LIN {X 0,Y 361.852,Z 288.032,A -85,B 0,C 180,E1 -12933.467,E2 -12933.467} C_VEL
LIN {X 0,Y 361.859,Z 288.029,A -85,B 0,C 180,E1 -12937.142,E2 -12937.142} C_VEL
LIN {X 0,Y 361.84,Z 288.029,A -85,B 0,C 180,E1 -12940.72,E2 -12940.72} C_VEL
LIN {X 0,Y 361.875,Z 288.032,A -85,B 0,C 180,E1 -12943.063,E2 -12943.063} C_VEL
LIN {X 0,Y 361.997,Z 288.011,A -85,B 0,C 180,E1 -12946.528,E2 -12946.528} C_VEL
LIN {X 0,Y 361.996,Z 288.014,A -85,B 0,C 180,E1 -12949.937,E2 -12949.937} C_VEL
LIN {X 0,Y 362.116,Z 288.001,A -85,B 0,C 180,E1 -12953.313,E2 -12953.313} C_VEL
LIN {X 0,Y 362.269,Z 287.981,A -85,B 0,C 180,E1 -12957.776,E2 -12957.776} C_VEL
LIN {X 0,Y 362.265,Z 287.979,A -85,B 0,C 180,E1 -12962.224,E2 -12962.224} C_VEL
LIN {X 0,Y 362.122,Z 287.997,A -85,B 0,C 180,E1 -12966.687,E2 -12966.687} C_VEL
LIN {X 0,Y 361.998,Z 288.011,A -85,B 0,C 180,E1 -12970.063,E2 -12970.063} C_VEL
LIN {X 0,Y 361.996,Z 288.018,A -85,B 0,C 180,E1 -12973.899,E2 -12973.899} C_VEL
LIN {X 0,Y 361.966,Z 288.024,A -85,B 0,C 180,E1 -12977.939,E2 -12977.939} C_VEL
LIN {X 0,Y 361.89,Z 288.034,A -85,B 0,C 180,E1 -12981.653,E2 -12981.653} C_VEL
LIN {X 0,Y 361.889,Z 288.003,A -85,B 0,C 180,E1 -12985.293,E2 -12985.293} C_VEL
LIN {X 0,Y 361.853,Z 288.035,A -85,B 0,C 180,E1 -12989.074,E2 -12989.074} C_VEL
LIN {X 0,Y 361.848,Z 288.021,A -85,B 0,C 180,E1 -12992.945,E2 -12992.945} C_VEL
LIN {X 0,Y 361.866,Z 288.032,A -85,B 0,C 180,E1 -12995.637,E2 -12995.637} C_VEL
LIN {X 0,Y 361.868,Z 288.029,A -85,B 0,C 180,E1 -12999.027,E2 -12999.027} C_VEL
LIN {X 0,Y 361.834,Z 288.037,A -85,B 0,C 180,E1 -13002.829,E2 -13002.829} C_VEL
LIN {X 0,Y 361.816,Z 288.04,A -85,B 0,C 180,E1 -13005.947,E2 -13005.947} C_VEL
LIN {X 0,Y 361.833,Z 288.027,A -85,B 0,C 180,E1 -13009.245,E2 -13009.245} C_VEL
LIN {X 0,Y 361.889,Z 288.094,A -85,B 0,C 180,E1 -13012.392,E2 -13012.392} C_VEL
LIN {X 0,Y 365.714,Z 301.841,A -85,B 0,C 180,E1 -13015.724,E2 -13015.724} C_VEL
LIN {X 0,Y 368.692,Z 314.163,A -85,B 0,C 180,E1 -13018.496,E2 -13018.496} C_VEL
LIN {X 0,Y 373.915,Z 326.027,A -85,B 0,C 180,E1 -13019.24,E2 -13019.24} C_VEL
LIN {X 0,Y 378.235,Z 348.319,A -85,B 0,C 180,E1 -13020.103,E2 -13020.103} C_VEL
LIN {X 0,Y 380.008,Z 359.01,A -85,B 0,C 180,E1 -13020.482,E2 -13020.482} C_VEL
LIN {X 0,Y 377.135,Z 474.361,A -85,B 0,C 180,E1 -13022.685,E2 -13022.685} C_VEL
LIN {X 0,Y 376.476,Z 489.459,A -85,B 0,C 180,E1 -13023.084,E2 -13023.084} C_VEL
LIN {X 0,Y 375.293,Z 504.296,A -85,B 0,C 180,E1 -13023.667,E2 -13023.667} C_VEL
LIN {X 0,Y 373.914,Z 518.628,A -85,B 0,C 180,E1 -13024.448,E2 -13024.448} C_VEL
LIN {X 0,Y 372.271,Z 532.938,A -85,B 0,C 180,E1 -13025.46,E2 -13025.46} C_VEL
LIN {X 0,Y 370.448,Z 546.556,A -85,B 0,C 180,E1 -13026.67,E2 -13026.67} C_VEL
LIN {X 0,Y 368.467,Z 560.156,A -85,B 0,C 180,E1 -13028.165,E2 -13028.165} C_VEL
LIN {X 0,Y 366.598,Z 572.399,A -85,B 0,C 180,E1 -13029.814,E2 -13029.814} C_VEL
LIN {X 0,Y 365.088,Z 582.684,A -85,B 0,C 180,E1 -13031.481,E2 -13031.481} C_VEL
LIN {X 0,Y 363.559,Z 592.741,A -85,B 0,C 180,E1 -13033.434,E2 -13033.434} C_VEL
LIN {X 0,Y 362.328,Z 601.099,A -85,B 0,C 180,E1 -13035.395,E2 -13035.395} C_VEL
LIN {X 0,Y 361.424,Z 608.963,A -85,B 0,C 180,E1 -13037.65,E2 -13037.65} C_VEL
LIN {X 0,Y 360.752,Z 615.222,A -85,B 0,C 180,E1 -13039.902,E2 -13039.902} C_VEL
LIN {X 0,Y 360.48,Z 620.073,A -85,B 0,C 180,E1 -13042.157,E2 -13042.157} C_VEL
LIN {X 0,Y 360.329,Z 623.628,A -85,B 0,C 180,E1 -13044.404,E2 -13044.404} C_VEL
LIN {X 0,Y 360.296,Z 625.968,A -85,B 0,C 180,E1 -13046.646,E2 -13046.646} C_VEL
LIN {X 0,Y 360.383,Z 627.148,A -85,B 0,C 180,E1 -13048.883,E2 -13048.883} C_VEL
LIN {X 0,Y 360.383,Z 627.145,A -85,B 0,C 180,E1 -13051.118,E2 -13051.118} C_VEL
LIN {X 0,Y 360.296,Z 625.956,A -85,B 0,C 180,E1 -13053.355,E2 -13053.355} C_VEL
LIN {X 0,Y 360.328,Z 623.608,A -85,B 0,C 180,E1 -13055.597,E2 -13055.597} C_VEL
LIN {X 0,Y 360.48,Z 620.052,A -85,B 0,C 180,E1 -13057.844,E2 -13057.844} C_VEL
LIN {X 0,Y 360.749,Z 615.196,A -85,B 0,C 180,E1 -13060.099,E2 -13060.099} C_VEL
LIN {X 0,Y 361.423,Z 608.921,A -85,B 0,C 180,E1 -13062.352,E2 -13062.352} C_VEL
LIN {X 0,Y 362.329,Z 601.044,A -85,B 0,C 180,E1 -13064.606,E2 -13064.606} C_VEL
LIN {X 0,Y 363.521,Z 592.679,A -85,B 0,C 180,E1 -13066.569,E2 -13066.569} C_VEL
LIN {X 0,Y 365.065,Z 582.609,A -85,B 0,C 180,E1 -13068.521,E2 -13068.521} C_VEL
LIN {X 0,Y 366.603,Z 572.317,A -85,B 0,C 180,E1 -13070.187,E2 -13070.187} C_VEL
LIN {X 0,Y 368.464,Z 560.062,A -85,B 0,C 180,E1 -13071.836,E2 -13071.836} C_VEL
LIN {X 0,Y 370.427,Z 546.423,A -85,B 0,C 180,E1 -13073.332,E2 -13073.332} C_VEL
LIN {X 0,Y 372.259,Z 532.757,A -85,B 0,C 180,E1 -13074.542,E2 -13074.542} C_VEL
LIN {X 0,Y 373.867,Z 518.7,A -85,B 0,C 180,E1 -13075.537,E2 -13075.537} C_VEL
LIN {X 0,Y 375.225,Z 504.036,A -85,B 0,C 180,E1 -13076.339,E2 -13076.339} C_VEL
LIN {X 0,Y 376.482,Z 488.055,A -85,B 0,C 180,E1 -13076.954,E2 -13076.954} C_VEL
LIN {X 0,Y 377.17,Z 472.026,A -85,B 0,C 180,E1 -13077.351,E2 -13077.351} C_VEL
LIN {X 0,Y 379.957,Z 359.045,A -85,B 0,C 180,E1 -13079.507,E2 -13079.507} C_VEL
LIN {X 0,Y 375.33,Z 332.928,A -85,B 0,C 180,E1 -13080.467,E2 -13080.467} C_VEL
LIN {X 0,Y 373.542,Z 325.186,A -85,B 0,C 180,E1 -13080.796,E2 -13080.796} C_VEL
LIN {X 0,Y 368.617,Z 313.906,A -85,B 0,C 180,E1 -13081.519,E2 -13081.519} C_VEL
LIN {X 0,Y 365.278,Z 300.144,A -85,B 0,C 180,E1 -13084.652,E2 -13084.652} C_VEL
LIN {X 0,Y 361.87,Z 288.032,A -85,B 0,C 180,E1 -13087.611,E2 -13087.611} C_VEL
LIN {X 0,Y 361.828,Z 288.038,A -85,B 0,C 180,E1 -13091.331,E2 -13091.331} C_VEL
LIN {X 0,Y 361.82,Z 288.042,A -85,B 0,C 180,E1 -13094.369,E2 -13094.369} C_VEL
LIN {X 0,Y 361.839,Z 288.032,A -85,B 0,C 180,E1 -13097.569,E2 -13097.569} C_VEL
LIN {X 0,Y 361.871,Z 288.033,A -85,B 0,C 180,E1 -13100.974,E2 -13100.974} C_VEL
LIN {X 0,Y 361.878,Z 288.027,A -85,B 0,C 180,E1 -13104.656,E2 -13104.656} C_VEL
LIN {X 0,Y 361.841,Z 288.034,A -85,B 0,C 180,E1 -13108.371,E2 -13108.371} C_VEL
LIN {X 0,Y 361.869,Z 288.027,A -85,B 0,C 180,E1 -13110.953,E2 -13110.953} C_VEL
LIN {X 0,Y 361.894,Z 288.028,A -85,B 0,C 180,E1 -13114.708,E2 -13114.708} C_VEL
LIN {X 0,Y 361.884,Z 288.031,A -85,B 0,C 180,E1 -13118.347,E2 -13118.347} C_VEL
LIN {X 0,Y 361.972,Z 288.02,A -85,B 0,C 180,E1 -13122.062,E2 -13122.062} C_VEL
LIN {X 0,Y 362.003,Z 288.018,A -85,B 0,C 180,E1 -13126.101,E2 -13126.101} C_VEL
LIN {X 0,Y 362.004,Z 288.015,A -85,B 0,C 180,E1 -13129.937,E2 -13129.937} C_VEL
LIN {X 0,Y 362.127,Z 287.993,A -85,B 0,C 180,E1 -13133.313,E2 -13133.313} C_VEL
LIN {X 0,Y 362.269,Z 287.978,A -85,B 0,C 180,E1 -13137.776,E2 -13137.776} C_VEL
LIN {X 0,Y 362.273,Z 287.979,A -85,B 0,C 180,E1 -13142.224,E2 -13142.224} C_VEL
LIN {X 0,Y 362.122,Z 287.996,A -85,B 0,C 180,E1 -13146.687,E2 -13146.687} C_VEL
LIN {X 0,Y 362.002,Z 288.01,A -85,B 0,C 180,E1 -13150.063,E2 -13150.063} C_VEL
LIN {X 0,Y 361.984,Z 288.014,A -85,B 0,C 180,E1 -13153.887,E2 -13153.887} C_VEL
LIN {X 0,Y 361.888,Z 288.026,A -85,B 0,C 180,E1 -13158.103,E2 -13158.103} C_VEL
LIN {X 0,Y 361.857,Z 288.033,A -85,B 0,C 180,E1 -13161.655,E2 -13161.655} C_VEL
LIN {X 0,Y 361.863,Z 288.036,A -85,B 0,C 180,E1 -13165.295,E2 -13165.295} C_VEL
LIN {X 0,Y 361.859,Z 288.016,A -85,B 0,C 180,E1 -13169.073,E2 -13169.073} C_VEL
LIN {X 0,Y 361.85,Z 288.033,A -85,B 0,C 180,E1 -13172.945,E2 -13172.945} C_VEL
LIN {X 0,Y 361.866,Z 288.03,A -85,B 0,C 180,E1 -13175.637,E2 -13175.637} C_VEL
LIN {X 0,Y 361.827,Z 288.035,A -85,B 0,C 180,E1 -13179.017,E2 -13179.017} C_VEL
LIN {X 0,Y 361.808,Z 288.04,A -85,B 0,C 180,E1 -13182.833,E2 -13182.833} C_VEL
LIN {X 0,Y 361.783,Z 288.04,A -85,B 0,C 180,E1 -13185.953,E2 -13185.953} C_VEL
LIN {X 0,Y 361.807,Z 288.045,A -85,B 0,C 180,E1 -13189.25,E2 -13189.25} C_VEL
LIN {X 0,Y 361.862,Z 288.026,A -85,B 0,C 180,E1 -13192.981,E2 -13192.981} C_VEL
LIN {X 0,Y 361.859,Z 288.031,A -85,B 0,C 180,E1 -13196.631,E2 -13196.631} C_VEL
LIN {X 0,Y 361.897,Z 288.144,A -85,B 0,C 180,E1 -13197.218,E2 -13197.218} C_VEL
LIN {X 0,Y 362.718,Z 291.26,A -85,B 0,C 180,E1 -13197.997,E2 -13197.997} C_VEL
LIN {X 0,Y 372.664,Z 310.987,A -85,B 0,C 180,E1 -13199.394,E2 -13199.394} C_VEL
LIN {X 0,Y 380.407,Z 328.591,A -85,B 0,C 180,E1 -13200.465,E2 -13200.465} C_VEL
LIN {X 0,Y 379.588,Z 366.53,A -85,B 0,C 180,E1 -13201.202,E2 -13201.202} C_VEL
LIN {X 0,Y 377.437,Z 452.401,A -85,B 0,C 180,E1 -13202.857,E2 -13202.857} C_VEL
LIN {X 0,Y 376.726,Z 467.883,A -85,B 0,C 180,E1 -13203.326,E2 -13203.326} C_VEL
LIN {X 0,Y 375.751,Z 482.572,A -85,B 0,C 180,E1 -13203.987,E2 -13203.987} C_VEL
LIN {X 0,Y 374.619,Z 495.263,A -85,B 0,C 180,E1 -13204.735,E2 -13204.735} C_VEL
LIN {X 0,Y 373.023,Z 509.629,A -85,B 0,C 180,E1 -13205.808,E2 -13205.808} C_VEL
LIN {X 0,Y 371.391,Z 522.676,A -85,B 0,C 180,E1 -13207.026,E2 -13207.026} C_VEL
LIN {X 0,Y 369.63,Z 534.686,A -85,B 0,C 180,E1 -13208.383,E2 -13208.383} C_VEL
LIN {X 0,Y 368.032,Z 545.767,A -85,B 0,C 180,E1 -13209.895,E2 -13209.895} C_VEL
LIN {X 0,Y 366.395,Z 555.931,A -85,B 0,C 180,E1 -13211.548,E2 -13211.548} C_VEL
LIN {X 0,Y 364.768,Z 565.873,A -85,B 0,C 180,E1 -13213.489,E2 -13213.489} C_VEL
LIN {X 0,Y 363.445,Z 574.112,A -85,B 0,C 180,E1 -13215.44,E2 -13215.44} C_VEL
LIN {X 0,Y 362.652,Z 580.052,A -85,B 0,C 180,E1 -13217.122,E2 -13217.122} C_VEL
LIN {X 0,Y 361.699,Z 586.588,A -85,B 0,C 180,E1 -13219.362,E2 -13219.362} C_VEL
LIN {X 0,Y 361.071,Z 591.693,A -85,B 0,C 180,E1 -13221.605,E2 -13221.605} C_VEL
LIN {X 0,Y 360.746,Z 594.97,A -85,B 0,C 180,E1 -13223.503,E2 -13223.503} C_VEL
LIN {X 0,Y 360.527,Z 597.508,A -85,B 0,C 180,E1 -13225.527,E2 -13225.527} C_VEL
LIN {X 0,Y 360.438,Z 599.238,A -85,B 0,C 180,E1 -13227.765,E2 -13227.765} C_VEL
LIN {X 0,Y 360.424,Z 599.842,A -85,B 0,C 180,E1 -13229.999,E2 -13229.999} C_VEL
LIN {X 0,Y 360.438,Z 599.283,A -85,B 0,C 180,E1 -13232.234,E2 -13232.234} C_VEL
LIN {X 0,Y 360.525,Z 597.615,A -85,B 0,C 180,E1 -13234.472,E2 -13234.472} C_VEL
LIN {X 0,Y 360.784,Z 594.793,A -85,B 0,C 180,E1 -13236.711,E2 -13236.711} C_VEL
LIN {X 0,Y 361.187,Z 590.754,A -85,B 0,C 180,E1 -13238.955,E2 -13238.955} C_VEL
LIN {X 0,Y 361.862,Z 585.393,A -85,B 0,C 180,E1 -13241.199,E2 -13241.199} C_VEL
LIN {X 0,Y 362.886,Z 578.554,A -85,B 0,C 180,E1 -13243.438,E2 -13243.438} C_VEL
LIN {X 0,Y 363.092,Z 577.022,A -85,B 0,C 180,E1 -13243.869,E2 -13243.869} C_VEL
LIN {X 0,Y 362.866,Z 574.172,A -85,B 0,C 180,E1 -13244.685,E2 -13244.685} C_VEL
LIN {X 0,Y 360.839,Z 569.392,A -85,B 0,C 180,E1 -13246.027,E2 -13246.027} C_VEL
LIN {X 0,Y 358.939,Z 564.173,A -85,B 0,C 180,E1 -13247.335,E2 -13247.335} C_VEL
LIN {X 0,Y 358.904,Z 560.595,A -85,B 0,C 180,E1 -13248.084,E2 -13248.084} C_VEL
LIN {X 0,Y 360.653,Z 550.211,A -85,B 0,C 180,E1 -13249.939,E2 -13249.939} C_VEL
LIN {X 0,Y 362.498,Z 538.889,A -85,B 0,C 180,E1 -13251.614,E2 -13251.614} C_VEL
LIN {X 0,Y 364.198,Z 527.692,A -85,B 0,C 180,E1 -13253.002,E2 -13253.002} C_VEL
LIN {X 0,Y 366.083,Z 514.164,A -85,B 0,C 180,E1 -13254.377,E2 -13254.377} C_VEL
LIN {X 0,Y 367.699,Z 500.855,A -85,B 0,C 180,E1 -13255.47,E2 -13255.47} C_VEL
LIN {X 0,Y 369.111,Z 486.646,A -85,B 0,C 180,E1 -13256.394,E2 -13256.394} C_VEL
LIN {X 0,Y 370.245,Z 471.515,A -85,B 0,C 180,E1 -13257.139,E2 -13257.139} C_VEL
LIN {X 0,Y 371.021,Z 456.576,A -85,B 0,C 180,E1 -13257.651,E2 -13257.651} C_VEL
LIN {X 0,Y 372.564,Z 404.124,A -85,B 0,C 180,E1 -13258.693,E2 -13258.693} C_VEL
LIN {X 0,Y 374.345,Z 330.704,A -85,B 0,C 180,E1 -13260.129,E2 -13260.129} C_VEL
LIN {X 0,Y 366.381,Z 312.908,A -85,B 0,C 180,E1 -13261.261,E2 -13261.261} C_VEL
LIN {X 0,Y 357.036,Z 294.502,A -85,B 0,C 180,E1 -13262.616,E2 -13262.616} C_VEL
LIN {X 0,Y 355.423,Z 291.234,A -85,B 0,C 180,E1 -13262.877,E2 -13262.877} C_VEL
LIN {X 0,Y 354.826,Z 288.912,A -85,B 0,C 180,E1 -13263.553,E2 -13263.553} C_VEL
LIN {X 0,Y 354.79,Z 288.911,A -85,B 0,C 180,E1 -13266.46,E2 -13266.46} C_VEL
LIN {X 0,Y 354.767,Z 288.92,A -85,B 0,C 180,E1 -13269.412,E2 -13269.412} C_VEL
LIN {X 0,Y 354.779,Z 288.904,A -85,B 0,C 180,E1 -13272.865,E2 -13272.865} C_VEL
LIN {X 0,Y 354.761,Z 288.919,A -85,B 0,C 180,E1 -13276.102,E2 -13276.102} C_VEL
LIN {X 0,Y 354.76,Z 288.909,A -85,B 0,C 180,E1 -13279.175,E2 -13279.175} C_VEL
LIN {X 0,Y 354.795,Z 288.899,A -85,B 0,C 180,E1 -13282.404,E2 -13282.404} C_VEL
LIN {X 0,Y 354.805,Z 288.896,A -85,B 0,C 180,E1 -13284.94,E2 -13284.94} C_VEL
LIN {X 0,Y 354.774,Z 288.914,A -85,B 0,C 180,E1 -13288.41,E2 -13288.41} C_VEL
LIN {X 0,Y 354.786,Z 288.913,A -85,B 0,C 180,E1 -13291.613,E2 -13291.613} C_VEL
LIN {X 0,Y 354.799,Z 288.912,A -85,B 0,C 180,E1 -13295.419,E2 -13295.419} C_VEL
LIN {X 0,Y 354.816,Z 288.911,A -85,B 0,C 180,E1 -13299.112,E2 -13299.112} C_VEL
LIN {X 0,Y 354.842,Z 288.91,A -85,B 0,C 180,E1 -13302.717,E2 -13302.717} C_VEL
LIN {X 0,Y 354.938,Z 288.888,A -85,B 0,C 180,E1 -13306.254,E2 -13306.254} C_VEL
LIN {X 0,Y 354.952,Z 288.893,A -85,B 0,C 180,E1 -13309.735,E2 -13309.735} C_VEL
LIN {X 0,Y 355.082,Z 288.878,A -85,B 0,C 180,E1 -13313.18,E2 -13313.18} C_VEL
LIN {X 0,Y 355.231,Z 288.858,A -85,B 0,C 180,E1 -13317.732,E2 -13317.732} C_VEL
LIN {X 0,Y 355.17,Z 288.855,A -85,B 0,C 180,E1 -13321.134,E2 -13321.134} C_VEL
LIN {X 0,Y 355.228,Z 288.856,A -85,B 0,C 180,E1 -13322.268,E2 -13322.268} C_VEL
LIN {X 0,Y 355.087,Z 288.874,A -85,B 0,C 180,E1 -13326.82,E2 -13326.82} C_VEL
LIN {X 0,Y 354.954,Z 288.887,A -85,B 0,C 180,E1 -13330.265,E2 -13330.265} C_VEL
LIN {X 0,Y 354.941,Z 288.895,A -85,B 0,C 180,E1 -13334.019,E2 -13334.019} C_VEL
LIN {X 0,Y 354.921,Z 288.899,A -85,B 0,C 180,E1 -13338.108,E2 -13338.108} C_VEL
LIN {X 0,Y 354.832,Z 288.91,A -85,B 0,C 180,E1 -13342.106,E2 -13342.106} C_VEL
LIN {X 0,Y 354.821,Z 288.885,A -85,B 0,C 180,E1 -13345.833,E2 -13345.833} C_VEL
LIN {X 0,Y 354.797,Z 288.911,A -85,B 0,C 180,E1 -13349.684,E2 -13349.684} C_VEL
LIN {X 0,Y 354.829,Z 288.902,A -85,B 0,C 180,E1 -13353.682,E2 -13353.682} C_VEL
LIN {X 0,Y 354.796,Z 288.905,A -85,B 0,C 180,E1 -13356.46,E2 -13356.46} C_VEL
LIN {X 0,Y 354.822,Z 288.91,A -85,B 0,C 180,E1 -13359.424,E2 -13359.424} C_VEL
LIN {X 0,Y 354.786,Z 288.915,A -85,B 0,C 180,E1 -13362.867,E2 -13362.867} C_VEL
LIN {X 0,Y 354.765,Z 288.917,A -85,B 0,C 180,E1 -13366.104,E2 -13366.104} C_VEL
LIN {X 0,Y 354.785,Z 288.905,A -85,B 0,C 180,E1 -13369.179,E2 -13369.179} C_VEL
LIN {X 0,Y 354.845,Z 289.112,A -85,B 0,C 180,E1 -13371.808,E2 -13371.808} C_VEL
LIN {X 0,Y 358.586,Z 302.202,A -85,B 0,C 180,E1 -13375.088,E2 -13375.088} C_VEL
LIN {X 0,Y 361.369,Z 313.699,A -85,B 0,C 180,E1 -13377.778,E2 -13377.778} C_VEL
LIN {X 0,Y 368.184,Z 329.155,A -85,B 0,C 180,E1 -13378.782,E2 -13378.782} C_VEL
LIN {X 0,Y 372.22,Z 350.437,A -85,B 0,C 180,E1 -13379.621,E2 -13379.621} C_VEL
LIN {X 0,Y 373.814,Z 360.578,A -85,B 0,C 180,E1 -13379.982,E2 -13379.982} C_VEL
LIN {X 0,Y 370.724,Z 477.12,A -85,B 0,C 180,E1 -13382.249,E2 -13382.249} C_VEL
LIN {X 0,Y 369.884,Z 492.864,A -85,B 0,C 180,E1 -13382.717,E2 -13382.717} C_VEL
LIN {X 0,Y 368.546,Z 507.946,A -85,B 0,C 180,E1 -13383.376,E2 -13383.376} C_VEL
LIN {X 0,Y 367.036,Z 522.28,A -85,B 0,C 180,E1 -13384.231,E2 -13384.231} C_VEL
LIN {X 0,Y 365.329,Z 535.876,A -85,B 0,C 180,E1 -13385.266,E2 -13385.266} C_VEL
LIN {X 0,Y 363.521,Z 548.916,A -85,B 0,C 180,E1 -13386.501,E2 -13386.501} C_VEL
LIN {X 0,Y 361.428,Z 562.036,A -85,B 0,C 180,E1 -13388.018,E2 -13388.018} C_VEL
LIN {X 0,Y 359.654,Z 573.379,A -85,B 0,C 180,E1 -13389.615,E2 -13389.615} C_VEL
LIN {X 0,Y 358.053,Z 583.935,A -85,B 0,C 180,E1 -13391.4,E2 -13391.4} C_VEL
LIN {X 0,Y 356.463,Z 593.733,A -85,B 0,C 180,E1 -13393.389,E2 -13393.389} C_VEL
LIN {X 0,Y 355.233,Z 601.993,A -85,B 0,C 180,E1 -13395.412,E2 -13395.412} C_VEL
LIN {X 0,Y 354.407,Z 608.691,A -85,B 0,C 180,E1 -13397.401,E2 -13397.401} C_VEL
LIN {X 0,Y 353.699,Z 614.95,A -85,B 0,C 180,E1 -13399.699,E2 -13399.699} C_VEL
LIN {X 0,Y 353.421,Z 619.802,A -85,B 0,C 180,E1 -13401.999,E2 -13401.999} C_VEL
LIN {X 0,Y 353.26,Z 623.358,A -85,B 0,C 180,E1 -13404.292,E2 -13404.292} C_VEL
LIN {X 0,Y 353.216,Z 625.698,A -85,B 0,C 180,E1 -13406.578,E2 -13406.578} C_VEL
LIN {X 0,Y 353.284,Z 626.877,A -85,B 0,C 180,E1 -13408.861,E2 -13408.861} C_VEL
LIN {X 0,Y 353.284,Z 626.875,A -85,B 0,C 180,E1 -13411.14,E2 -13411.14} C_VEL
LIN {X 0,Y 353.216,Z 625.685,A -85,B 0,C 180,E1 -13413.423,E2 -13413.423} C_VEL
LIN {X 0,Y 353.276,Z 623.08,A -85,B 0,C 180,E1 -13415.909,E2 -13415.909} C_VEL
LIN {X 0,Y 353.456,Z 618.698,A -85,B 0,C 180,E1 -13418.577,E2 -13418.577} C_VEL
LIN {X 0,Y 353.887,Z 613.48,A -85,B 0,C 180,E1 -13420.875,E2 -13420.875} C_VEL
LIN {X 0,Y 354.642,Z 606.815,A -85,B 0,C 180,E1 -13423.174,E2 -13423.174} C_VEL
LIN {X 0,Y 355.546,Z 599.642,A -85,B 0,C 180,E1 -13425.184,E2 -13425.184} C_VEL
LIN {X 0,Y 356.833,Z 591.038,A -85,B 0,C 180,E1 -13427.184,E2 -13427.184} C_VEL
LIN {X 0,Y 358.546,Z 580.695,A -85,B 0,C 180,E1 -13429.168,E2 -13429.168} C_VEL
LIN {X 0,Y 360.175,Z 570.118,A -85,B 0,C 180,E1 -13430.862,E2 -13430.862} C_VEL
LIN {X 0,Y 362.011,Z 558.63,A -85,B 0,C 180,E1 -13432.396,E2 -13432.396} C_VEL
LIN {X 0,Y 363.885,Z 546.147,A -85,B 0,C 180,E1 -13433.778,E2 -13433.778} C_VEL
LIN {X 0,Y 365.782,Z 532.481,A -85,B 0,C 180,E1 -13435.006,E2 -13435.006} C_VEL
LIN {X 0,Y 367.42,Z 518.711,A -85,B 0,C 180,E1 -13435.997,E2 -13435.997} C_VEL
LIN {X 0,Y 368.874,Z 503.758,A -85,B 0,C 180,E1 -13436.828,E2 -13436.828} C_VEL
LIN {X 0,Y 370.143,Z 487.771,A -85,B 0,C 180,E1 -13437.455,E2 -13437.455} C_VEL
LIN {X 0,Y 370.885,Z 471.735,A -85,B 0,C 180,E1 -13437.855,E2 -13437.855} C_VEL
LIN {X 0,Y 373.771,Z 360.404,A -85,B 0,C 180,E1 -13440.009,E2 -13440.009} C_VEL
LIN {X 0,Y 369.837,Z 337.692,A -85,B 0,C 180,E1 -13440.858,E2 -13440.858} C_VEL
LIN {X 0,Y 367.838,Z 328.195,A -85,B 0,C 180,E1 -13441.254,E2 -13441.254} C_VEL
LIN {X 0,Y 361.346,Z 313.573,A -85,B 0,C 180,E1 -13442.231,E2 -13442.231} C_VEL
LIN {X 0,Y 358.258,Z 301.022,A -85,B 0,C 180,E1 -13445.177,E2 -13445.177} C_VEL
LIN {X 0,Y 354.844,Z 288.909,A -85,B 0,C 180,E1 -13448.239,E2 -13448.239} C_VEL
LIN {X 0,Y 354.796,Z 288.914,A -85,B 0,C 180,E1 -13452.338,E2 -13452.338} C_VEL
LIN {X 0,Y 354.769,Z 288.907,A -85,B 0,C 180,E1 -13456.104,E2 -13456.104} C_VEL
LIN {X 0,Y 354.791,Z 288.914,A -85,B 0,C 180,E1 -13459.18,E2 -13459.18} C_VEL
LIN {X 0,Y 354.81,Z 288.91,A -85,B 0,C 180,E1 -13462.403,E2 -13462.403} C_VEL
LIN {X 0,Y 354.815,Z 288.907,A -85,B 0,C 180,E1 -13464.941,E2 -13464.941} C_VEL
LIN {X 0,Y 354.797,Z 288.911,A -85,B 0,C 180,E1 -13468.406,E2 -13468.406} C_VEL
LIN {X 0,Y 354.806,Z 288.908,A -85,B 0,C 180,E1 -13471.615,E2 -13471.615} C_VEL
LIN {X 0,Y 354.855,Z 288.904,A -85,B 0,C 180,E1 -13475.423,E2 -13475.423} C_VEL
LIN {X 0,Y 354.831,Z 288.908,A -85,B 0,C 180,E1 -13479.114,E2 -13479.114} C_VEL
LIN {X 0,Y 354.903,Z 288.901,A -85,B 0,C 180,E1 -13482.72,E2 -13482.72} C_VEL
LIN {X 0,Y 354.956,Z 288.897,A -85,B 0,C 180,E1 -13486.255,E2 -13486.255} C_VEL
LIN {X 0,Y 354.96,Z 288.89,A -85,B 0,C 180,E1 -13489.736,E2 -13489.736} C_VEL
LIN {X 0,Y 355.092,Z 288.868,A -85,B 0,C 180,E1 -13493.18,E2 -13493.18} C_VEL
LIN {X 0,Y 355.231,Z 288.854,A -85,B 0,C 180,E1 -13497.732,E2 -13497.732} C_VEL
LIN {X 0,Y 355.15,Z 288.867,A -85,B 0,C 180,E1 -13501.134,E2 -13501.134} C_VEL
LIN {X 0,Y 355.236,Z 288.856,A -85,B 0,C 180,E1 -13502.268,E2 -13502.268} C_VEL
LIN {X 0,Y 355.088,Z 288.872,A -85,B 0,C 180,E1 -13506.82,E2 -13506.82} C_VEL
LIN {X 0,Y 354.958,Z 288.886,A -85,B 0,C 180,E1 -13510.265,E2 -13510.265} C_VEL
LIN {X 0,Y 354.928,Z 288.892,A -85,B 0,C 180,E1 -13514.006,E2 -13514.006} C_VEL
LIN {X 0,Y 354.846,Z 288.903,A -85,B 0,C 180,E1 -13518.068,E2 -13518.068} C_VEL
LIN {X 0,Y 354.81,Z 288.907,A -85,B 0,C 180,E1 -13522.108,E2 -13522.108} C_VEL
LIN {X 0,Y 354.802,Z 288.908,A -85,B 0,C 180,E1 -13525.835,E2 -13525.835} C_VEL
LIN {X 0,Y 354.796,Z 288.903,A -85,B 0,C 180,E1 -13529.684,E2 -13529.684} C_VEL
LIN {X 0,Y 354.789,Z 288.912,A -85,B 0,C 180,E1 -13532.333,E2 -13532.333} C_VEL
LIN {X 0,Y 354.821,Z 288.907,A -85,B 0,C 180,E1 -13535.698,E2 -13535.698} C_VEL
LIN {X 0,Y 354.771,Z 288.915,A -85,B 0,C 180,E1 -13539.412,E2 -13539.412} C_VEL
LIN {X 0,Y 354.763,Z 288.918,A -85,B 0,C 180,E1 -13542.862,E2 -13542.862} C_VEL
LIN {X 0,Y 354.733,Z 288.918,A -85,B 0,C 180,E1 -13546.097,E2 -13546.097} C_VEL
LIN {X 0,Y 354.758,Z 288.922,A -85,B 0,C 180,E1 -13549.174,E2 -13549.174} C_VEL
LIN {X 0,Y 354.8,Z 288.907,A -85,B 0,C 180,E1 -13552.404,E2 -13552.404} C_VEL
LIN {X 0,Y 354.81,Z 288.911,A -85,B 0,C 180,E1 -13554.94,E2 -13554.94} C_VEL
LIN {X 0,Y 354.85,Z 289.016,A -85,B 0,C 180,E1 -13556.624,E2 -13556.624} C_VEL
LIN {X 0,Y 355.598,Z 291.578,A -85,B 0,C 180,E1 -13557.277,E2 -13557.277} C_VEL
LIN {X 0,Y 366.442,Z 312.982,A -85,B 0,C 180,E1 -13558.855,E2 -13558.855} C_VEL
LIN {X 0,Y 374.33,Z 330.792,A -85,B 0,C 180,E1 -13559.978,E2 -13559.978} C_VEL
LIN {X 0,Y 372.099,Z 418.657,A -85,B 0,C 180,E1 -13561.687,E2 -13561.687} C_VEL
LIN {X 0,Y 371.037,Z 455.65,A -85,B 0,C 180,E1 -13562.426,E2 -13562.426} C_VEL
LIN {X 0,Y 370.215,Z 471.175,A -85,B 0,C 180,E1 -13562.947,E2 -13562.947} C_VEL
LIN {X 0,Y 369.208,Z 485.293,A -85,B 0,C 180,E1 -13563.633,E2 -13563.633} C_VEL
LIN {X 0,Y 367.832,Z 499.494,A -85,B 0,C 180,E1 -13564.538,E2 -13564.538} C_VEL
LIN {X 0,Y 366.176,Z 513.055,A -85,B 0,C 180,E1 -13565.628,E2 -13565.628} C_VEL
LIN {X 0,Y 364.255,Z 526.808,A -85,B 0,C 180,E1 -13567.001,E2 -13567.001} C_VEL
LIN {X 0,Y 362.546,Z 538.145,A -85,B 0,C 180,E1 -13568.387,E2 -13568.387} C_VEL
LIN {X 0,Y 360.706,Z 549.584,A -85,B 0,C 180,E1 -13570.063,E2 -13570.063} C_VEL
LIN {X 0,Y 359.13,Z 559.203,A -85,B 0,C 180,E1 -13571.753,E2 -13571.753} C_VEL
LIN {X 0,Y 357.508,Z 568.629,A -85,B 0,C 180,E1 -13573.731,E2 -13573.731} C_VEL
LIN {X 0,Y 356.307,Z 576.467,A -85,B 0,C 180,E1 -13575.726,E2 -13575.726} C_VEL
LIN {X 0,Y 355.091,Z 583.784,A -85,B 0,C 180,E1 -13578.005,E2 -13578.005} C_VEL
LIN {X 0,Y 354.34,Z 589.582,A -85,B 0,C 180,E1 -13580.294,E2 -13580.294} C_VEL
LIN {X 0,Y 353.919,Z 593.013,A -85,B 0,C 180,E1 -13582.009,E2 -13582.009} C_VEL
LIN {X 0,Y 353.599,Z 596.486,A -85,B 0,C 180,E1 -13584.296,E2 -13584.296} C_VEL
LIN {X 0,Y 353.352,Z 598.785,A -85,B 0,C 180,E1 -13586.579,E2 -13586.579} C_VEL
LIN {X 0,Y 353.324,Z 599.956,A -85,B 0,C 180,E1 -13588.86,E2 -13588.86} C_VEL
LIN {X 0,Y 353.324,Z 599.971,A -85,B 0,C 180,E1 -13591.139,E2 -13591.139} C_VEL
LIN {X 0,Y 353.351,Z 598.861,A -85,B 0,C 180,E1 -13593.42,E2 -13593.42} C_VEL
LIN {X 0,Y 353.596,Z 596.62,A -85,B 0,C 180,E1 -13595.703,E2 -13595.703} C_VEL
LIN {X 0,Y 353.901,Z 593.202,A -85,B 0,C 180,E1 -13597.99,E2 -13597.99} C_VEL
LIN {X 0,Y 354.488,Z 588.516,A -85,B 0,C 180,E1 -13600.278,E2 -13600.278} C_VEL
LIN {X 0,Y 355.336,Z 582.442,A -85,B 0,C 180,E1 -13602.565,E2 -13602.565} C_VEL
LIN {X 0,Y 356.328,Z 575.837,A -85,B 0,C 180,E1 -13604.564,E2 -13604.564} C_VEL
LIN {X 0,Y 357.662,Z 567.847,A -85,B 0,C 180,E1 -13606.554,E2 -13606.554} C_VEL
LIN {X 0,Y 358.904,Z 560.595,A -85,B 0,C 180,E1 -13608.084,E2 -13608.084} C_VEL
LIN {X 0,Y 358.894,Z 556.949,A -85,B 0,C 180,E1 -13608.821,E2 -13608.821} C_VEL
LIN {X 0,Y 355.779,Z 545.813,A -85,B 0,C 180,E1 -13611.017,E2 -13611.017} C_VEL
LIN {X 0,Y 355.531,Z 541.648,A -85,B 0,C 180,E1 -13611.691,E2 -13611.691} C_VEL
LIN {X 0,Y 355.714,Z 540.173,A -85,B 0,C 180,E1 -13611.899,E2 -13611.899} C_VEL
LIN {X 0,Y 357.461,Z 529.137,A -85,B 0,C 180,E1 -13613.308,E2 -13613.308} C_VEL
LIN {X 0,Y 359.417,Z 515.884,A -85,B 0,C 180,E1 -13614.706,E2 -13614.706} C_VEL
LIN {X 0,Y 361.099,Z 502.882,A -85,B 0,C 180,E1 -13615.815,E2 -13615.815} C_VEL
LIN {X 0,Y 362.465,Z 490.066,A -85,B 0,C 180,E1 -13616.698,E2 -13616.698} C_VEL
LIN {X 0,Y 363.705,Z 475.109,A -85,B 0,C 180,E1 -13617.497,E2 -13617.497} C_VEL
LIN {X 0,Y 364.62,Z 460.242,A -85,B 0,C 180,E1 -13618.062,E2 -13618.062} C_VEL
LIN {X 0,Y 365.282,Z 442.705,A -85,B 0,C 180,E1 -13618.475,E2 -13618.475} C_VEL
LIN {X 0,Y 368.22,Z 333.905,A -85,B 0,C 180,E1 -13620.618,E2 -13620.618} C_VEL
LIN {X 0,Y 367.995,Z 332.244,A -85,B 0,C 180,E1 -13620.676,E2 -13620.676} C_VEL
LIN {X 0,Y 360.065,Z 314.543,A -85,B 0,C 180,E1 -13621.842,E2 -13621.842} C_VEL
LIN {X 0,Y 351.227,Z 297.376,A -85,B 0,C 180,E1 -13623.161,E2 -13623.161} C_VEL
LIN {X 0,Y 348.21,Z 291.481,A -85,B 0,C 180,E1 -13623.663,E2 -13623.663} C_VEL
LIN {X 0,Y 347.754,Z 289.798,A -85,B 0,C 180,E1 -13624.201,E2 -13624.201} C_VEL
LIN {X 0,Y 347.753,Z 289.797,A -85,B 0,C 180,E1 -13627.321,E2 -13627.321} C_VEL
LIN {X 0,Y 347.694,Z 289.799,A -85,B 0,C 180,E1 -13630.302,E2 -13630.302} C_VEL
LIN {X 0,Y 347.719,Z 289.783,A -85,B 0,C 180,E1 -13633.408,E2 -13633.408} C_VEL
LIN {X 0,Y 347.721,Z 289.785,A -85,B 0,C 180,E1 -13636.687,E2 -13636.687} C_VEL
LIN {X 0,Y 347.698,Z 289.797,A -85,B 0,C 180,E1 -13640.182,E2 -13640.182} C_VEL
LIN {X 0,Y 347.751,Z 289.771,A -85,B 0,C 180,E1 -13642.678,E2 -13642.678} C_VEL
LIN {X 0,Y 347.746,Z 289.788,A -85,B 0,C 180,E1 -13645.956,E2 -13645.956} C_VEL
LIN {X 0,Y 347.727,Z 289.792,A -85,B 0,C 180,E1 -13649.65,E2 -13649.65} C_VEL
LIN {X 0,Y 347.73,Z 289.791,A -85,B 0,C 180,E1 -13653.599,E2 -13653.599} C_VEL
LIN {X 0,Y 347.745,Z 289.788,A -85,B 0,C 180,E1 -13656.159,E2 -13656.159} C_VEL
LIN {X 0,Y 347.763,Z 289.79,A -85,B 0,C 180,E1 -13659.906,E2 -13659.906} C_VEL
LIN {X 0,Y 347.787,Z 289.787,A -85,B 0,C 180,E1 -13663.566,E2 -13663.566} C_VEL
LIN {X 0,Y 347.885,Z 289.773,A -85,B 0,C 180,E1 -13667.16,E2 -13667.16} C_VEL
LIN {X 0,Y 347.932,Z 289.759,A -85,B 0,C 180,E1 -13670.7,E2 -13670.7} C_VEL
LIN {X 0,Y 348.035,Z 289.756,A -85,B 0,C 180,E1 -13674.205,E2 -13674.205} C_VEL
LIN {X 0,Y 348.193,Z 289.734,A -85,B 0,C 180,E1 -13677.686,E2 -13677.686} C_VEL
LIN {X 0,Y 348.139,Z 289.731,A -85,B 0,C 180,E1 -13681.157,E2 -13681.157} C_VEL
LIN {X 0,Y 348.189,Z 289.733,A -85,B 0,C 180,E1 -13682.313,E2 -13682.313} C_VEL
LIN {X 0,Y 348.054,Z 289.75,A -85,B 0,C 180,E1 -13686.959,E2 -13686.959} C_VEL
LIN {X 0,Y 347.894,Z 289.765,A -85,B 0,C 180,E1 -13690.475,E2 -13690.475} C_VEL
LIN {X 0,Y 347.897,Z 289.77,A -85,B 0,C 180,E1 -13694.15,E2 -13694.15} C_VEL
LIN {X 0,Y 347.889,Z 289.773,A -85,B 0,C 180,E1 -13698.29,E2 -13698.29} C_VEL
LIN {X 0,Y 347.787,Z 289.791,A -85,B 0,C 180,E1 -13701.635,E2 -13701.635} C_VEL
LIN {X 0,Y 347.771,Z 289.76,A -85,B 0,C 180,E1 -13705.111,E2 -13705.111} C_VEL
LIN {X 0,Y 347.737,Z 289.789,A -85,B 0,C 180,E1 -13707.7,E2 -13707.7} C_VEL
LIN {X 0,Y 347.738,Z 289.784,A -85,B 0,C 180,E1 -13710.349,E2 -13710.349} C_VEL
LIN {X 0,Y 347.746,Z 289.789,A -85,B 0,C 180,E1 -13714.044,E2 -13714.044} C_VEL
LIN {X 0,Y 347.76,Z 289.773,A -85,B 0,C 180,E1 -13717.321,E2 -13717.321} C_VEL
LIN {X 0,Y 347.731,Z 289.794,A -85,B 0,C 180,E1 -13720.297,E2 -13720.297} C_VEL
LIN {X 0,Y 347.721,Z 289.794,A -85,B 0,C 180,E1 -13723.408,E2 -13723.408} C_VEL
LIN {X 0,Y 347.723,Z 289.792,A -85,B 0,C 180,E1 -13726.687,E2 -13726.687} C_VEL
LIN {X 0,Y 347.745,Z 289.787,A -85,B 0,C 180,E1 -13730.173,E2 -13730.173} C_VEL
LIN {X 0,Y 347.791,Z 289.809,A -85,B 0,C 180,E1 -13731.121,E2 -13731.121} C_VEL
LIN {X 0,Y 351.584,Z 303.182,A -85,B 0,C 180,E1 -13734.571,E2 -13734.571} C_VEL
LIN {X 0,Y 354.071,Z 313.378,A -85,B 0,C 180,E1 -13737.03,E2 -13737.03} C_VEL
LIN {X 0,Y 362.3,Z 331.558,A -85,B 0,C 180,E1 -13738.277,E2 -13738.277} C_VEL
LIN {X 0,Y 366.074,Z 351.444,A -85,B 0,C 180,E1 -13739.083,E2 -13739.083} C_VEL
LIN {X 0,Y 367.651,Z 361.718,A -85,B 0,C 180,E1 -13739.457,E2 -13739.457} C_VEL
LIN {X 0,Y 364.463,Z 476.867,A -85,B 0,C 180,E1 -13741.729,E2 -13741.729} C_VEL
LIN {X 0,Y 363.599,Z 492.605,A -85,B 0,C 180,E1 -13742.205,E2 -13742.205} C_VEL
LIN {X 0,Y 362.193,Z 507.682,A -85,B 0,C 180,E1 -13742.872,E2 -13742.872} C_VEL
LIN {X 0,Y 360.68,Z 521.765,A -85,B 0,C 180,E1 -13743.723,E2 -13743.723} C_VEL
LIN {X 0,Y 358.868,Z 535.609,A -85,B 0,C 180,E1 -13744.79,E2 -13744.79} C_VEL
LIN {X 0,Y 356.946,Z 548.646,A -85,B 0,C 180,E1 -13746.041,E2 -13746.041} C_VEL
LIN {X 0,Y 354.843,Z 561.768,A -85,B 0,C 180,E1 -13747.588,E2 -13747.588} C_VEL
LIN {X 0,Y 352.951,Z 573.067,A -85,B 0,C 180,E1 -13749.203,E2 -13749.203} C_VEL
LIN {X 0,Y 351.243,Z 583.663,A -85,B 0,C 180,E1 -13751.026,E2 -13751.026} C_VEL
LIN {X 0,Y 349.595,Z 593.461,A -85,B 0,C 180,E1 -13753.053,E2 -13753.053} C_VEL
LIN {X 0,Y 348.296,Z 601.645,A -85,B 0,C 180,E1 -13755.093,E2 -13755.093} C_VEL
LIN {X 0,Y 347.405,Z 608.418,A -85,B 0,C 180,E1 -13757.143,E2 -13757.143} C_VEL
LIN {X 0,Y 346.657,Z 614.679,A -85,B 0,C 180,E1 -13759.487,E2 -13759.487} C_VEL
LIN {X 0,Y 346.345,Z 619.531,A -85,B 0,C 180,E1 -13761.834,E2 -13761.834} C_VEL
LIN {X 0,Y 346.179,Z 623.087,A -85,B 0,C 180,E1 -13764.175,E2 -13764.175} C_VEL
LIN {X 0,Y 346.138,Z 625.428,A -85,B 0,C 180,E1 -13766.508,E2 -13766.508} C_VEL
LIN {X 0,Y 346.185,Z 626.607,A -85,B 0,C 180,E1 -13768.837,E2 -13768.837} C_VEL
LIN {X 0,Y 346.185,Z 626.604,A -85,B 0,C 180,E1 -13771.164,E2 -13771.164} C_VEL
LIN {X 0,Y 346.138,Z 625.415,A -85,B 0,C 180,E1 -13773.493,E2 -13773.493} C_VEL
LIN {X 0,Y 346.196,Z 622.992,A -85,B 0,C 180,E1 -13775.885,E2 -13775.885} C_VEL
LIN {X 0,Y 346.329,Z 619.506,A -85,B 0,C 180,E1 -13778.167,E2 -13778.167} C_VEL
LIN {X 0,Y 346.654,Z 614.648,A -85,B 0,C 180,E1 -13780.514,E2 -13780.514} C_VEL
LIN {X 0,Y 347.406,Z 608.371,A -85,B 0,C 180,E1 -13782.858,E2 -13782.858} C_VEL
LIN {X 0,Y 348.442,Z 600.493,A -85,B 0,C 180,E1 -13785.202,E2 -13785.202} C_VEL
LIN {X 0,Y 349.767,Z 592.127,A -85,B 0,C 180,E1 -13787.241,E2 -13787.241} C_VEL
LIN {X 0,Y 351.504,Z 582.059,A -85,B 0,C 180,E1 -13789.263,E2 -13789.263} C_VEL
LIN {X 0,Y 353.18,Z 571.766,A -85,B 0,C 180,E1 -13790.989,E2 -13790.989} C_VEL
LIN {X 0,Y 355.214,Z 559.51,A -85,B 0,C 180,E1 -13792.695,E2 -13792.695} C_VEL
LIN {X 0,Y 357.339,Z 545.87,A -85,B 0,C 180,E1 -13794.241,E2 -13794.241} C_VEL
LIN {X 0,Y 359.315,Z 532.203,A -85,B 0,C 180,E1 -13795.488,E2 -13795.488} C_VEL
LIN {X 0,Y 360.979,Z 518.816,A -85,B 0,C 180,E1 -13796.468,E2 -13796.468} C_VEL
LIN {X 0,Y 362.543,Z 503.479,A -85,B 0,C 180,E1 -13797.335,E2 -13797.335} C_VEL
LIN {X 0,Y 363.87,Z 487.488,A -85,B 0,C 180,E1 -13797.969,E2 -13797.969} C_VEL
LIN {X 0,Y 364.615,Z 471.444,A -85,B 0,C 180,E1 -13798.376,E2 -13798.376} C_VEL
LIN {X 0,Y 367.597,Z 361.496,A -85,B 0,C 180,E1 -13800.536,E2 -13800.536} C_VEL
LIN {X 0,Y 363.956,Z 340.064,A -85,B 0,C 180,E1 -13801.353,E2 -13801.353} C_VEL
LIN {X 0,Y 362.033,Z 331.007,A -85,B 0,C 180,E1 -13801.743,E2 -13801.743} C_VEL
LIN {X 0,Y 357.127,Z 320.151,A -85,B 0,C 180,E1 -13802.478,E2 -13802.478} C_VEL
LIN {X 0,Y 354.067,Z 313.266,A -85,B 0,C 180,E1 -13802.973,E2 -13802.973} C_VEL
LIN {X 0,Y 351.187,Z 301.767,A -85,B 0,C 180,E1 -13805.76,E2 -13805.76} C_VEL
LIN {X 0,Y 347.775,Z 289.781,A -85,B 0,C 180,E1 -13808.883,E2 -13808.883} C_VEL
LIN {X 0,Y 347.752,Z 289.79,A -85,B 0,C 180,E1 -13811.831,E2 -13811.831} C_VEL
LIN {X 0,Y 347.708,Z 289.797,A -85,B 0,C 180,E1 -13815.027,E2 -13815.027} C_VEL
LIN {X 0,Y 347.753,Z 289.794,A -85,B 0,C 180,E1 -13818.398,E2 -13818.398} C_VEL
LIN {X 0,Y 347.776,Z 289.786,A -85,B 0,C 180,E1 -13822.012,E2 -13822.012} C_VEL
LIN {X 0,Y 347.748,Z 289.788,A -85,B 0,C 180,E1 -13825.537,E2 -13825.537} C_VEL
LIN {X 0,Y 347.749,Z 289.788,A -85,B 0,C 180,E1 -13828.301,E2 -13828.301} C_VEL
LIN {X 0,Y 347.75,Z 289.786,A -85,B 0,C 180,E1 -13830.985,E2 -13830.985} C_VEL
LIN {X 0,Y 347.759,Z 289.784,A -85,B 0,C 180,E1 -13833.602,E2 -13833.602} C_VEL
LIN {X 0,Y 347.774,Z 289.786,A -85,B 0,C 180,E1 -13836.161,E2 -13836.161} C_VEL
LIN {X 0,Y 347.811,Z 289.784,A -85,B 0,C 180,E1 -13839.909,E2 -13839.909} C_VEL
LIN {X 0,Y 347.871,Z 289.779,A -85,B 0,C 180,E1 -13842.36,E2 -13842.36} C_VEL
LIN {X 0,Y 347.902,Z 289.772,A -85,B 0,C 180,E1 -13845.971,E2 -13845.971} C_VEL
LIN {X 0,Y 347.9,Z 289.767,A -85,B 0,C 180,E1 -13849.525,E2 -13849.525} C_VEL
LIN {X 0,Y 348.059,Z 289.744,A -85,B 0,C 180,E1 -13853.042,E2 -13853.042} C_VEL
LIN {X 0,Y 348.193,Z 289.73,A -85,B 0,C 180,E1 -13857.687,E2 -13857.687} C_VEL
LIN {X 0,Y 348.122,Z 289.742,A -85,B 0,C 180,E1 -13861.157,E2 -13861.157} C_VEL
LIN {X 0,Y 348.197,Z 289.733,A -85,B 0,C 180,E1 -13862.314,E2 -13862.314} C_VEL
LIN {X 0,Y 348.056,Z 289.748,A -85,B 0,C 180,E1 -13866.959,E2 -13866.959} C_VEL
LIN {X 0,Y 347.898,Z 289.765,A -85,B 0,C 180,E1 -13870.475,E2 -13870.475} C_VEL
LIN {X 0,Y 347.884,Z 289.768,A -85,B 0,C 180,E1 -13874.137,E2 -13874.137} C_VEL
LIN {X 0,Y 347.797,Z 289.78,A -85,B 0,C 180,E1 -13878.241,E2 -13878.241} C_VEL
LIN {X 0,Y 347.767,Z 289.789,A -85,B 0,C 180,E1 -13881.624,E2 -13881.624} C_VEL
LIN {X 0,Y 347.741,Z 289.795,A -85,B 0,C 180,E1 -13885.114,E2 -13885.114} C_VEL
LIN {X 0,Y 347.727,Z 289.771,A -85,B 0,C 180,E1 -13887.701,E2 -13887.701} C_VEL
LIN {X 0,Y 347.739,Z 289.791,A -85,B 0,C 180,E1 -13890.349,E2 -13890.349} C_VEL
LIN {X 0,Y 347.752,Z 289.792,A -85,B 0,C 180,E1 -13894.043,E2 -13894.043} C_VEL
LIN {X 0,Y 347.757,Z 289.792,A -85,B 0,C 180,E1 -13897.322,E2 -13897.322} C_VEL
LIN {X 0,Y 347.698,Z 289.796,A -85,B 0,C 180,E1 -13900.302,E2 -13900.302} C_VEL
LIN {X 0,Y 347.71,Z 289.794,A -85,B 0,C 180,E1 -13903.41,E2 -13903.41} C_VEL
LIN {X 0,Y 347.684,Z 289.798,A -85,B 0,C 180,E1 -13906.694,E2 -13906.694} C_VEL
LIN {X 0,Y 347.702,Z 289.796,A -85,B 0,C 180,E1 -13910.182,E2 -13910.182} C_VEL
LIN {X 0,Y 347.756,Z 289.782,A -85,B 0,C 180,E1 -13912.678,E2 -13912.678} C_VEL
LIN {X 0,Y 347.769,Z 289.862,A -85,B 0,C 180,E1 -13915.987,E2 -13915.987} C_VEL
LIN {X 0,Y 348.374,Z 291.832,A -85,B 0,C 180,E1 -13916.507,E2 -13916.507} C_VEL
LIN {X 0,Y 359.996,Z 314.451,A -85,B 0,C 180,E1 -13918.259,E2 -13918.259} C_VEL
LIN {X 0,Y 368.145,Z 332.6,A -85,B 0,C 180,E1 -13919.454,E2 -13919.454} C_VEL
LIN {X 0,Y 365.857,Z 419.16,A -85,B 0,C 180,E1 -13921.164,E2 -13921.164} C_VEL
LIN {X 0,Y 364.779,Z 455.937,A -85,B 0,C 180,E1 -13921.912,E2 -13921.912} C_VEL
LIN {X 0,Y 363.909,Z 471.512,A -85,B 0,C 180,E1 -13922.441,E2 -13922.441} C_VEL
LIN {X 0,Y 362.814,Z 486.274,A -85,B 0,C 180,E1 -13923.175,E2 -13923.175} C_VEL
LIN {X 0,Y 361.455,Z 499.77,A -85,B 0,C 180,E1 -13924.056,E2 -13924.056} C_VEL
LIN {X 0,Y 359.719,Z 513.331,A -85,B 0,C 180,E1 -13925.161,E2 -13925.161} C_VEL
LIN {X 0,Y 357.743,Z 527.082,A -85,B 0,C 180,E1 -13926.557,E2 -13926.557} C_VEL
LIN {X 0,Y 355.948,Z 538.42,A -85,B 0,C 180,E1 -13927.966,E2 -13927.966} C_VEL
LIN {X 0,Y 354.02,Z 549.858,A -85,B 0,C 180,E1 -13929.67,E2 -13929.67} C_VEL
LIN {X 0,Y 352.349,Z 559.478,A -85,B 0,C 180,E1 -13931.389,E2 -13931.389} C_VEL
LIN {X 0,Y 350.671,Z 568.903,A -85,B 0,C 180,E1 -13933.405,E2 -13933.405} C_VEL
LIN {X 0,Y 349.379,Z 576.741,A -85,B 0,C 180,E1 -13935.436,E2 -13935.436} C_VEL
LIN {X 0,Y 348.433,Z 582.39,A -85,B 0,C 180,E1 -13937.18,E2 -13937.18} C_VEL
LIN {X 0,Y 347.51,Z 588.539,A -85,B 0,C 180,E1 -13939.512,E2 -13939.512} C_VEL
LIN {X 0,Y 346.86,Z 593.286,A -85,B 0,C 180,E1 -13941.846,E2 -13941.846} C_VEL
LIN {X 0,Y 346.518,Z 596.758,A -85,B 0,C 180,E1 -13944.179,E2 -13944.179} C_VEL
LIN {X 0,Y 346.274,Z 599.056,A -85,B 0,C 180,E1 -13946.509,E2 -13946.509} C_VEL
LIN {X 0,Y 346.229,Z 600.226,A -85,B 0,C 180,E1 -13948.836,E2 -13948.836} C_VEL
LIN {X 0,Y 346.229,Z 600.241,A -85,B 0,C 180,E1 -13951.163,E2 -13951.163} C_VEL
LIN {X 0,Y 346.273,Z 599.13,A -85,B 0,C 180,E1 -13953.49,E2 -13953.49} C_VEL
LIN {X 0,Y 346.515,Z 596.891,A -85,B 0,C 180,E1 -13955.82,E2 -13955.82} C_VEL
LIN {X 0,Y 346.843,Z 593.473,A -85,B 0,C 180,E1 -13958.154,E2 -13958.154} C_VEL
LIN {X 0,Y 347.477,Z 588.787,A -85,B 0,C 180,E1 -13960.488,E2 -13960.488} C_VEL
LIN {X 0,Y 348.4,Z 582.711,A -85,B 0,C 180,E1 -13962.82,E2 -13962.82} C_VEL
LIN {X 0,Y 349.434,Z 575.86,A -85,B 0,C 180,E1 -13964.932,E2 -13964.932} C_VEL
LIN {X 0,Y 351.089,Z 566.887,A -85,B 0,C 180,E1 -13967.173,E2 -13967.173} C_VEL
LIN {X 0,Y 352.838,Z 557.041,A -85,B 0,C 180,E1 -13969.187,E2 -13969.187} C_VEL
LIN {X 0,Y 354.867,Z 545.45,A -85,B 0,C 180,E1 -13971.129,E2 -13971.129} C_VEL
LIN {X 0,Y 355.714,Z 540.173,A -85,B 0,C 180,E1 -13971.899,E2 -13971.899} C_VEL
LIN {X 0,Y 355.847,Z 535.817,A -85,B 0,C 180,E1 -13972.527,E2 -13972.527} C_VEL
LIN {X 0,Y 354.335,Z 528.678,A -85,B 0,C 180,E1 -13973.604,E2 -13973.604} C_VEL
LIN {X 0,Y 352.84,Z 521.18,A -85,B 0,C 180,E1 -13974.637,E2 -13974.637} C_VEL
LIN {X 0,Y 352.979,Z 516.234,A -85,B 0,C 180,E1 -13975.178,E2 -13975.178} C_VEL
LIN {X 0,Y 354.734,Z 503.145,A -85,B 0,C 180,E1 -13976.314,E2 -13976.314} C_VEL
LIN {X 0,Y 356.154,Z 490.328,A -85,B 0,C 180,E1 -13977.21,E2 -13977.21} C_VEL
LIN {X 0,Y 357.44,Z 475.22,A -85,B 0,C 180,E1 -13978.029,E2 -13978.029} C_VEL
LIN {X 0,Y 358.443,Z 459.358,A -85,B 0,C 180,E1 -13978.629,E2 -13978.629} C_VEL
LIN {X 0,Y 359.268,Z 437.589,A -85,B 0,C 180,E1 -13979.117,E2 -13979.117} C_VEL
LIN {X 0,Y 362.093,Z 335.919,A -85,B 0,C 180,E1 -13981.153,E2 -13981.153} C_VEL
LIN {X 0,Y 361.86,Z 334.195,A -85,B 0,C 180,E1 -13981.215,E2 -13981.215} C_VEL
LIN {X 0,Y 353.98,Z 316.712,A -85,B 0,C 180,E1 -13982.41,E2 -13982.41} C_VEL
LIN {X 0,Y 344.67,Z 298.743,A -85,B 0,C 180,E1 -13983.849,E2 -13983.849} C_VEL
LIN {X 0,Y 340.963,Z 291.86,A -85,B 0,C 180,E1 -13984.463,E2 -13984.463} C_VEL
LIN {X 0,Y 340.695,Z 290.676,A -85,B 0,C 180,E1 -13984.85,E2 -13984.85} C_VEL
LIN {X 0,Y 340.691,Z 290.673,A -85,B 0,C 180,E1 -13988.382,E2 -13988.382} C_VEL
LIN {X 0,Y 340.689,Z 290.666,A -85,B 0,C 180,E1 -13992.043,E2 -13992.043} C_VEL
LIN {X 0,Y 340.648,Z 290.673,A -85,B 0,C 180,E1 -13996.227,E2 -13996.227} C_VEL
LIN {X 0,Y 340.666,Z 290.657,A -85,B 0,C 180,E1 -13998.687,E2 -13998.687} C_VEL
LIN {X 0,Y 340.715,Z 290.664,A -85,B 0,C 180,E1 -14001.77,E2 -14001.77} C_VEL
LIN {X 0,Y 340.72,Z 290.662,A -85,B 0,C 180,E1 -14005.596,E2 -14005.596} C_VEL
LIN {X 0,Y 340.68,Z 290.668,A -85,B 0,C 180,E1 -14008.953,E2 -14008.953} C_VEL
LIN {X 0,Y 340.684,Z 290.666,A -85,B 0,C 180,E1 -14012.504,E2 -14012.504} C_VEL
LIN {X 0,Y 340.712,Z 290.667,A -85,B 0,C 180,E1 -14015.635,E2 -14015.635} C_VEL
LIN {X 0,Y 340.704,Z 290.669,A -85,B 0,C 180,E1 -14019.471,E2 -14019.471} C_VEL
LIN {X 0,Y 340.755,Z 290.655,A -85,B 0,C 180,E1 -14021.978,E2 -14021.978} C_VEL
LIN {X 0,Y 340.83,Z 290.645,A -85,B 0,C 180,E1 -14025.73,E2 -14025.73} C_VEL
LIN {X 0,Y 340.844,Z 290.65,A -85,B 0,C 180,E1 -14029.305,E2 -14029.305} C_VEL
LIN {X 0,Y 340.997,Z 290.634,A -85,B 0,C 180,E1 -14032.896,E2 -14032.896} C_VEL
LIN {X 0,Y 340.818,Z 290.648,A -85,B 0,C 180,E1 -14035.269,E2 -14035.269} C_VEL
LIN {X 0,Y 341.154,Z 290.611,A -85,B 0,C 180,E1 -14037.639,E2 -14037.639} C_VEL
LIN {X 0,Y 341.108,Z 290.607,A -85,B 0,C 180,E1 -14041.18,E2 -14041.18} C_VEL
LIN {X 0,Y 341.127,Z 290.613,A -85,B 0,C 180,E1 -14042.361,E2 -14042.361} C_VEL
LIN {X 0,Y 341.015,Z 290.622,A -85,B 0,C 180,E1 -14045.914,E2 -14045.914} C_VEL
LIN {X 0,Y 340.961,Z 290.639,A -85,B 0,C 180,E1 -14048.356,E2 -14048.356} C_VEL
LIN {X 0,Y 340.848,Z 290.647,A -85,B 0,C 180,E1 -14051.899,E2 -14051.899} C_VEL
LIN {X 0,Y 340.818,Z 290.647,A -85,B 0,C 180,E1 -14055.549,E2 -14055.549} C_VEL
LIN {X 0,Y 340.835,Z 290.65,A -85,B 0,C 180,E1 -14058.466,E2 -14058.466} C_VEL
LIN {X 0,Y 340.752,Z 290.667,A -85,B 0,C 180,E1 -14061.857,E2 -14061.857} C_VEL
LIN {X 0,Y 340.722,Z 290.638,A -85,B 0,C 180,E1 -14065.668,E2 -14065.668} C_VEL
LIN {X 0,Y 340.706,Z 290.666,A -85,B 0,C 180,E1 -14069.674,E2 -14069.674} C_VEL
LIN {X 0,Y 340.687,Z 290.65,A -85,B 0,C 180,E1 -14072.436,E2 -14072.436} C_VEL
LIN {X 0,Y 340.716,Z 290.67,A -85,B 0,C 180,E1 -14075.279,E2 -14075.279} C_VEL
LIN {X 0,Y 340.708,Z 290.656,A -85,B 0,C 180,E1 -14078.386,E2 -14078.386} C_VEL
LIN {X 0,Y 340.697,Z 290.673,A -85,B 0,C 180,E1 -14082.046,E2 -14082.046} C_VEL
LIN {X 0,Y 340.65,Z 290.675,A -85,B 0,C 180,E1 -14086.227,E2 -14086.227} C_VEL
LIN {X 0,Y 340.686,Z 290.662,A -85,B 0,C 180,E1 -14089.753,E2 -14089.753} C_VEL
LIN {X 0,Y 340.76,Z 290.85,A -85,B 0,C 180,E1 -14090.485,E2 -14090.485} C_VEL
LIN {X 0,Y 344.492,Z 303.818,A -85,B 0,C 180,E1 -14093.943,E2 -14093.943} C_VEL
LIN {X 0,Y 346.809,Z 313.084,A -85,B 0,C 180,E1 -14096.248,E2 -14096.248} C_VEL
LIN {X 0,Y 356.464,Z 334.171,A -85,B 0,C 180,E1 -14097.762,E2 -14097.762} C_VEL
LIN {X 0,Y 360.107,Z 353.41,A -85,B 0,C 180,E1 -14098.563,E2 -14098.563} C_VEL
LIN {X 0,Y 361.496,Z 362.819,A -85,B 0,C 180,E1 -14098.91,E2 -14098.91} C_VEL
LIN {X 0,Y 358.171,Z 478.12,A -85,B 0,C 180,E1 -14101.227,E2 -14101.227} C_VEL
LIN {X 0,Y 357.244,Z 493.26,A -85,B 0,C 180,E1 -14101.707,E2 -14101.707} C_VEL
LIN {X 0,Y 355.89,Z 507.419,A -85,B 0,C 180,E1 -14102.35,E2 -14102.35} C_VEL
LIN {X 0,Y 354.338,Z 521.227,A -85,B 0,C 180,E1 -14103.194,E2 -14103.194} C_VEL
LIN {X 0,Y 352.429,Z 535.342,A -85,B 0,C 180,E1 -14104.296,E2 -14104.296} C_VEL
LIN {X 0,Y 350.44,Z 548.378,A -85,B 0,C 180,E1 -14105.567,E2 -14105.567} C_VEL
LIN {X 0,Y 348.431,Z 560.423,A -85,B 0,C 180,E1 -14106.996,E2 -14106.996} C_VEL
LIN {X 0,Y 346.48,Z 571.587,A -85,B 0,C 180,E1 -14108.586,E2 -14108.586} C_VEL
LIN {X 0,Y 344.72,Z 581.87,A -85,B 0,C 180,E1 -14110.343,E2 -14110.343} C_VEL
LIN {X 0,Y 342.962,Z 591.926,A -85,B 0,C 180,E1 -14112.407,E2 -14112.407} C_VEL
LIN {X 0,Y 341.515,Z 600.283,A -85,B 0,C 180,E1 -14114.483,E2 -14114.483} C_VEL
LIN {X 0,Y 340.414,Z 608.146,A -85,B 0,C 180,E1 -14116.874,E2 -14116.874} C_VEL
LIN {X 0,Y 339.618,Z 614.407,A -85,B 0,C 180,E1 -14119.267,E2 -14119.267} C_VEL
LIN {X 0,Y 339.265,Z 619.259,A -85,B 0,C 180,E1 -14121.663,E2 -14121.663} C_VEL
LIN {X 0,Y 339.087,Z 622.983,A -85,B 0,C 180,E1 -14124.187,E2 -14124.187} C_VEL
LIN {X 0,Y 339.061,Z 625.158,A -85,B 0,C 180,E1 -14126.435,E2 -14126.435} C_VEL
LIN {X 0,Y 339.086,Z 626.336,A -85,B 0,C 180,E1 -14128.813,E2 -14128.813} C_VEL
LIN {X 0,Y 339.137,Z 626.493,A -85,B 0,C 180,E1 -14130.001,E2 -14130.001} C_VEL
LIN {X 0,Y 339.026,Z 625.881,A -85,B 0,C 180,E1 -14132.377,E2 -14132.377} C_VEL
LIN {X 0,Y 339.044,Z 624.116,A -85,B 0,C 180,E1 -14134.757,E2 -14134.757} C_VEL
LIN {X 0,Y 339.138,Z 621.169,A -85,B 0,C 180,E1 -14137.143,E2 -14137.143} C_VEL
LIN {X 0,Y 339.39,Z 616.973,A -85,B 0,C 180,E1 -14139.536,E2 -14139.536} C_VEL
LIN {X 0,Y 340.019,Z 611.425,A -85,B 0,C 180,E1 -14141.929,E2 -14141.929} C_VEL
LIN {X 0,Y 340.875,Z 604.369,A -85,B 0,C 180,E1 -14144.325,E2 -14144.325} C_VEL
LIN {X 0,Y 342.285,Z 595.606,A -85,B 0,C 180,E1 -14146.706,E2 -14146.706} C_VEL
LIN {X 0,Y 343.9,Z 586.306,A -85,B 0,C 180,E1 -14148.777,E2 -14148.777} C_VEL
LIN {X 0,Y 345.521,Z 576.905,A -85,B 0,C 180,E1 -14150.532,E2 -14150.532} C_VEL
LIN {X 0,Y 347.65,Z 564.61,A -85,B 0,C 180,E1 -14152.432,E2 -14152.432} C_VEL
LIN {X 0,Y 349.813,Z 552.132,A -85,B 0,C 180,E1 -14154.007,E2 -14154.007} C_VEL
LIN {X 0,Y 351.712,Z 539.862,A -85,B 0,C 180,E1 -14155.286,E2 -14155.286} C_VEL
LIN {X 0,Y 353.636,Z 526.454,A -85,B 0,C 180,E1 -14156.417,E2 -14156.417} C_VEL
LIN {X 0,Y 355.37,Z 512.121,A -85,B 0,C 180,E1 -14157.375,E2 -14157.375} C_VEL
LIN {X 0,Y 356.781,Z 497.882,A -85,B 0,C 180,E1 -14158.094,E2 -14158.094} C_VEL
LIN {X 0,Y 357.912,Z 482.634,A -85,B 0,C 180,E1 -14158.637,E2 -14158.637} C_VEL
LIN {X 0,Y 358.722,Z 458.613,A -85,B 0,C 180,E1 -14159.167,E2 -14159.167} C_VEL
LIN {X 0,Y 361.422,Z 361.832,A -85,B 0,C 180,E1 -14161.101,E2 -14161.101} C_VEL
LIN {X 0,Y 357.245,Z 337.796,A -85,B 0,C 180,E1 -14162.056,E2 -14162.056} C_VEL
LIN {X 0,Y 356.067,Z 333.272,A -85,B 0,C 180,E1 -14162.279,E2 -14162.279} C_VEL
LIN {X 0,Y 347.643,Z 315.056,A -85,B 0,C 180,E1 -14163.59,E2 -14163.59} C_VEL
LIN {X 0,Y 346.806,Z 312.955,A -85,B 0,C 180,E1 -14163.752,E2 -14163.752} C_VEL
LIN {X 0,Y 344.205,Z 302.738,A -85,B 0,C 180,E1 -14166.309,E2 -14166.309} C_VEL
LIN {X 0,Y 340.724,Z 290.656,A -85,B 0,C 180,E1 -14169.571,E2 -14169.571} C_VEL
LIN {X 0,Y 340.678,Z 290.674,A -85,B 0,C 180,E1 -14172.905,E2 -14172.905} C_VEL
LIN {X 0,Y 340.678,Z 290.662,A -85,B 0,C 180,E1 -14177.096,E2 -14177.096} C_VEL
LIN {X 0,Y 340.702,Z 290.669,A -85,B 0,C 180,E1 -14180.248,E2 -14180.248} C_VEL
LIN {X 0,Y 340.713,Z 290.667,A -85,B 0,C 180,E1 -14183.56,E2 -14183.56} C_VEL
LIN {X 0,Y 340.698,Z 290.67,A -85,B 0,C 180,E1 -14186.154,E2 -14186.154} C_VEL
LIN {X 0,Y 340.727,Z 290.661,A -85,B 0,C 180,E1 -14190.034,E2 -14190.034} C_VEL
LIN {X 0,Y 340.727,Z 290.661,A -85,B 0,C 180,E1 -14193.014,E2 -14193.014} C_VEL
LIN {X 0,Y 340.746,Z 290.663,A -85,B 0,C 180,E1 -14195.638,E2 -14195.638} C_VEL
LIN {X 0,Y 340.741,Z 290.665,A -85,B 0,C 180,E1 -14199.474,E2 -14199.474} C_VEL
LIN {X 0,Y 340.862,Z 290.648,A -85,B 0,C 180,E1 -14201.985,E2 -14201.985} C_VEL
LIN {X 0,Y 340.874,Z 290.644,A -85,B 0,C 180,E1 -14205.705,E2 -14205.705} C_VEL
LIN {X 0,Y 340.852,Z 290.644,A -85,B 0,C 180,E1 -14209.306,E2 -14209.306} C_VEL
LIN {X 0,Y 341.006,Z 290.622,A -85,B 0,C 180,E1 -14212.897,E2 -14212.897} C_VEL
LIN {X 0,Y 340.818,Z 290.656,A -85,B 0,C 180,E1 -14215.269,E2 -14215.269} C_VEL
LIN {X 0,Y 341.13,Z 290.61,A -85,B 0,C 180,E1 -14217.639,E2 -14217.639} C_VEL
LIN {X 0,Y 341.093,Z 290.617,A -85,B 0,C 180,E1 -14221.181,E2 -14221.181} C_VEL
LIN {X 0,Y 341.135,Z 290.612,A -85,B 0,C 180,E1 -14222.362,E2 -14222.362} C_VEL
LIN {X 0,Y 341.003,Z 290.627,A -85,B 0,C 180,E1 -14227.103,E2 -14227.103} C_VEL
LIN {X 0,Y 340.851,Z 290.643,A -85,B 0,C 180,E1 -14230.695,E2 -14230.695} C_VEL
LIN {X 0,Y 340.823,Z 290.647,A -85,B 0,C 180,E1 -14234.327,E2 -14234.327} C_VEL
LIN {X 0,Y 340.759,Z 290.656,A -85,B 0,C 180,E1 -14238.424,E2 -14238.424} C_VEL
LIN {X 0,Y 340.722,Z 290.664,A -85,B 0,C 180,E1 -14241.841,E2 -14241.841} C_VEL
LIN {X 0,Y 340.674,Z 290.669,A -85,B 0,C 180,E1 -14245.672,E2 -14245.672} C_VEL
LIN {X 0,Y 340.678,Z 290.647,A -85,B 0,C 180,E1 -14248.325,E2 -14248.325} C_VEL
LIN {X 0,Y 340.696,Z 290.67,A -85,B 0,C 180,E1 -14251.045,E2 -14251.045} C_VEL
LIN {X 0,Y 340.718,Z 290.667,A -85,B 0,C 180,E1 -14255.279,E2 -14255.279} C_VEL
LIN {X 0,Y 340.696,Z 290.667,A -85,B 0,C 180,E1 -14258.382,E2 -14258.382} C_VEL
LIN {X 0,Y 340.665,Z 290.673,A -85,B 0,C 180,E1 -14262.038,E2 -14262.038} C_VEL
LIN {X 0,Y 340.619,Z 290.679,A -85,B 0,C 180,E1 -14265.45,E2 -14265.45} C_VEL
LIN {X 0,Y 340.636,Z 290.676,A -85,B 0,C 180,E1 -14268.682,E2 -14268.682} C_VEL
LIN {X 0,Y 340.72,Z 290.666,A -85,B 0,C 180,E1 -14271.77,E2 -14271.77} C_VEL
LIN {X 0,Y 340.732,Z 290.765,A -85,B 0,C 180,E1 -14275.339,E2 -14275.339} C_VEL
LIN {X 0,Y 341.064,Z 292.151,A -85,B 0,C 180,E1 -14275.69,E2 -14275.69} C_VEL
LIN {X 0,Y 347.901,Z 304.838,A -85,B 0,C 180,E1 -14276.771,E2 -14276.771} C_VEL
LIN {X 0,Y 355.814,Z 320.651,A -85,B 0,C 180,E1 -14277.982,E2 -14277.982} C_VEL
LIN {X 0,Y 362.013,Z 334.658,A -85,B 0,C 180,E1 -14278.92,E2 -14278.92} C_VEL
LIN {X 0,Y 359.742,Z 418.202,A -85,B 0,C 180,E1 -14280.598,E2 -14280.598} C_VEL
LIN {X 0,Y 358.559,Z 456.224,A -85,B 0,C 180,E1 -14281.38,E2 -14281.38} C_VEL
LIN {X 0,Y 357.633,Z 471.843,A -85,B 0,C 180,E1 -14281.918,E2 -14281.918} C_VEL
LIN {X 0,Y 356.456,Z 487.131,A -85,B 0,C 180,E1 -14282.697,E2 -14282.697} C_VEL
LIN {X 0,Y 355.086,Z 500.048,A -85,B 0,C 180,E1 -14283.555,E2 -14283.555} C_VEL
LIN {X 0,Y 353.299,Z 513.606,A -85,B 0,C 180,E1 -14284.678,E2 -14284.678} C_VEL
LIN {X 0,Y 351.248,Z 527.357,A -85,B 0,C 180,E1 -14286.097,E2 -14286.097} C_VEL
LIN {X 0,Y 349.349,Z 538.695,A -85,B 0,C 180,E1 -14287.527,E2 -14287.527} C_VEL
LIN {X 0,Y 347.37,Z 550.132,A -85,B 0,C 180,E1 -14289.263,E2 -14289.263} C_VEL
LIN {X 0,Y 345.604,Z 559.752,A -85,B 0,C 180,E1 -14291.012,E2 -14291.012} C_VEL
LIN {X 0,Y 343.855,Z 569.176,A -85,B 0,C 180,E1 -14293.066,E2 -14293.066} C_VEL
LIN {X 0,Y 342.455,Z 577.015,A -85,B 0,C 180,E1 -14295.135,E2 -14295.135} C_VEL
LIN {X 0,Y 341.508,Z 582.662,A -85,B 0,C 180,E1 -14296.916,E2 -14296.916} C_VEL
LIN {X 0,Y 340.492,Z 588.813,A -85,B 0,C 180,E1 -14299.294,E2 -14299.294} C_VEL
LIN {X 0,Y 339.808,Z 593.558,A -85,B 0,C 180,E1 -14301.675,E2 -14301.675} C_VEL
LIN {X 0,Y 339.443,Z 597.03,A -85,B 0,C 180,E1 -14304.057,E2 -14304.057} C_VEL
LIN {X 0,Y 339.199,Z 599.326,A -85,B 0,C 180,E1 -14306.436,E2 -14306.436} C_VEL
LIN {X 0,Y 339.134,Z 600.497,A -85,B 0,C 180,E1 -14308.812,E2 -14308.812} C_VEL
LIN {X 0,Y 339.134,Z 600.511,A -85,B 0,C 180,E1 -14311.187,E2 -14311.187} C_VEL
LIN {X 0,Y 339.198,Z 599.4,A -85,B 0,C 180,E1 -14313.563,E2 -14313.563} C_VEL
LIN {X 0,Y 339.442,Z 597.161,A -85,B 0,C 180,E1 -14315.942,E2 -14315.942} C_VEL
LIN {X 0,Y 339.795,Z 593.743,A -85,B 0,C 180,E1 -14318.324,E2 -14318.324} C_VEL
LIN {X 0,Y 340.457,Z 589.057,A -85,B 0,C 180,E1 -14320.706,E2 -14320.706} C_VEL
LIN {X 0,Y 341.473,Z 582.98,A -85,B 0,C 180,E1 -14323.084,E2 -14323.084} C_VEL
LIN {X 0,Y 342.719,Z 575.328,A -85,B 0,C 180,E1 -14325.461,E2 -14325.461} C_VEL
LIN {X 0,Y 344.287,Z 567.157,A -85,B 0,C 180,E1 -14327.523,E2 -14327.523} C_VEL
LIN {X 0,Y 346.117,Z 557.309,A -85,B 0,C 180,E1 -14329.574,E2 -14329.574} C_VEL
LIN {X 0,Y 348.186,Z 545.987,A -85,B 0,C 180,E1 -14331.511,E2 -14331.511} C_VEL
LIN {X 0,Y 350.132,Z 534.072,A -85,B 0,C 180,E1 -14333.198,E2 -14333.198} C_VEL
LIN {X 0,Y 352.207,Z 521.804,A -85,B 0,C 180,E1 -14334.616,E2 -14334.616} C_VEL
LIN {X 0,Y 352.979,Z 516.234,A -85,B 0,C 180,E1 -14335.178,E2 -14335.178} C_VEL
LIN {X 0,Y 353.126,Z 511.267,A -85,B 0,C 180,E1 -14335.696,E2 -14335.696} C_VEL
LIN {X 0,Y 351.624,Z 503.149,A -85,B 0,C 180,E1 -14336.588,E2 -14336.588} C_VEL
LIN {X 0,Y 350.072,Z 494.778,A -85,B 0,C 180,E1 -14337.414,E2 -14337.414} C_VEL
LIN {X 0,Y 349.975,Z 489.418,A -85,B 0,C 180,E1 -14337.816,E2 -14337.816} C_VEL
LIN {X 0,Y 351.238,Z 474.944,A -85,B 0,C 180,E1 -14338.598,E2 -14338.598} C_VEL
LIN {X 0,Y 352.253,Z 459.612,A -85,B 0,C 180,E1 -14339.18,E2 -14339.18} C_VEL
LIN {X 0,Y 353.092,Z 437.834,A -85,B 0,C 180,E1 -14339.677,E2 -14339.677} C_VEL
LIN {X 0,Y 356.016,Z 337.707,A -85,B 0,C 180,E1 -14341.71,E2 -14341.71} C_VEL
LIN {X 0,Y 355.578,Z 335.758,A -85,B 0,C 180,E1 -14341.8,E2 -14341.8} C_VEL
LIN {X 0,Y 347.467,Z 317.968,A -85,B 0,C 180,E1 -14343.071,E2 -14343.071} C_VEL
LIN {X 0,Y 338.033,Z 299.873,A -85,B 0,C 180,E1 -14344.585,E2 -14344.585} C_VEL
LIN {X 0,Y 333.945,Z 292.78,A -85,B 0,C 180,E1 -14345.258,E2 -14345.258} C_VEL
LIN {X 0,Y 333.769,Z 292.028,A -85,B 0,C 180,E1 -14345.355,E2 -14345.355} C_VEL
LIN {X 0,Y 333.656,Z 291.545,A -85,B 0,C 180,E1 -14345.513,E2 -14345.513} C_VEL
LIN {X 0,Y 333.618,Z 291.557,A -85,B 0,C 180,E1 -14349.196,E2 -14349.196} C_VEL
LIN {X 0,Y 333.624,Z 291.54,A -85,B 0,C 180,E1 -14352.498,E2 -14352.498} C_VEL
LIN {X 0,Y 333.592,Z 291.556,A -85,B 0,C 180,E1 -14355.954,E2 -14355.954} C_VEL
LIN {X 0,Y 333.599,Z 291.545,A -85,B 0,C 180,E1 -14359.324,E2 -14359.324} C_VEL
LIN {X 0,Y 333.659,Z 291.521,A -85,B 0,C 180,E1 -14363.169,E2 -14363.169} C_VEL
LIN {X 0,Y 333.67,Z 291.534,A -85,B 0,C 180,E1 -14365.341,E2 -14365.341} C_VEL
LIN {X 0,Y 333.619,Z 291.549,A -85,B 0,C 180,E1 -14368.22,E2 -14368.22} C_VEL
LIN {X 0,Y 333.626,Z 291.551,A -85,B 0,C 180,E1 -14371.02,E2 -14371.02} C_VEL
LIN {X 0,Y 333.654,Z 291.548,A -85,B 0,C 180,E1 -14374.922,E2 -14374.922} C_VEL
LIN {X 0,Y 333.647,Z 291.549,A -85,B 0,C 180,E1 -14379.017,E2 -14379.017} C_VEL
LIN {X 0,Y 333.707,Z 291.531,A -85,B 0,C 180,E1 -14381.584,E2 -14381.584} C_VEL
LIN {X 0,Y 333.772,Z 291.524,A -85,B 0,C 180,E1 -14385.6,E2 -14385.6} C_VEL
LIN {X 0,Y 333.814,Z 291.526,A -85,B 0,C 180,E1 -14389.077,E2 -14389.077} C_VEL
LIN {X 0,Y 333.953,Z 291.512,A -85,B 0,C 180,E1 -14392.746,E2 -14392.746} C_VEL
LIN {X 0,Y 333.784,Z 291.524,A -85,B 0,C 180,E1 -14395.169,E2 -14395.169} C_VEL
LIN {X 0,Y 334.091,Z 291.49,A -85,B 0,C 180,E1 -14397.589,E2 -14397.589} C_VEL
LIN {X 0,Y 334.076,Z 291.482,A -85,B 0,C 180,E1 -14401.205,E2 -14401.205} C_VEL
LIN {X 0,Y 333.809,Z 291.529,A -85,B 0,C 180,E1 -14403.621,E2 -14403.621} C_VEL
LIN {X 0,Y 333.988,Z 291.497,A -85,B 0,C 180,E1 -14406.039,E2 -14406.039} C_VEL
LIN {X 0,Y 333.818,Z 291.524,A -85,B 0,C 180,E1 -14409.696,E2 -14409.696} C_VEL
LIN {X 0,Y 333.795,Z 291.531,A -85,B 0,C 180,E1 -14413.391,E2 -14413.391} C_VEL
LIN {X 0,Y 333.745,Z 291.537,A -85,B 0,C 180,E1 -14417.146,E2 -14417.146} C_VEL
LIN {X 0,Y 333.735,Z 291.532,A -85,B 0,C 180,E1 -14419.69,E2 -14419.69} C_VEL
LIN {X 0,Y 333.689,Z 291.542,A -85,B 0,C 180,E1 -14422.278,E2 -14422.278} C_VEL
LIN {X 0,Y 333.69,Z 291.512,A -85,B 0,C 180,E1 -14425.091,E2 -14425.091} C_VEL
LIN {X 0,Y 333.653,Z 291.548,A -85,B 0,C 180,E1 -14428.977,E2 -14428.977} C_VEL
LIN {X 0,Y 333.644,Z 291.527,A -85,B 0,C 180,E1 -14432.588,E2 -14432.588} C_VEL
LIN {X 0,Y 333.674,Z 291.537,A -85,B 0,C 180,E1 -14436.139,E2 -14436.139} C_VEL
LIN {X 0,Y 333.645,Z 291.545,A -85,B 0,C 180,E1 -14439.192,E2 -14439.192} C_VEL
LIN {X 0,Y 333.631,Z 291.551,A -85,B 0,C 180,E1 -14442.5,E2 -14442.5} C_VEL
LIN {X 0,Y 333.595,Z 291.556,A -85,B 0,C 180,E1 -14445.955,E2 -14445.955} C_VEL
LIN {X 0,Y 333.658,Z 291.622,A -85,B 0,C 180,E1 -14449.74,E2 -14449.74} C_VEL
LIN {X 0,Y 337.45,Z 304.52,A -85,B 0,C 180,E1 -14453.304,E2 -14453.304} C_VEL
LIN {X 0,Y 339.569,Z 312.708,A -85,B 0,C 180,E1 -14455.424,E2 -14455.424} C_VEL
LIN {X 0,Y 350.318,Z 336.036,A -85,B 0,C 180,E1 -14457.176,E2 -14457.176} C_VEL
LIN {X 0,Y 351.316,Z 339.516,A -85,B 0,C 180,E1 -14457.363,E2 -14457.363} C_VEL
LIN {X 0,Y 355.103,Z 361.127,A -85,B 0,C 180,E1 -14458.253,E2 -14458.253} C_VEL
LIN {X 0,Y 355.402,Z 364.023,A -85,B 0,C 180,E1 -14458.35,E2 -14458.35} C_VEL
LIN {X 0,Y 351.902,Z 479.372,A -85,B 0,C 180,E1 -14460.706,E2 -14460.706} C_VEL
LIN {X 0,Y 350.843,Z 494.831,A -85,B 0,C 180,E1 -14461.224,E2 -14461.224} C_VEL
LIN {X 0,Y 349.322,Z 509.762,A -85,B 0,C 180,E1 -14461.948,E2 -14461.948} C_VEL
LIN {X 0,Y 347.448,Z 525.114,A -85,B 0,C 180,E1 -14462.959,E2 -14462.959} C_VEL
LIN {X 0,Y 345.292,Z 539.76,A -85,B 0,C 180,E1 -14464.211,E2 -14464.211} C_VEL
LIN {X 0,Y 343.093,Z 553.215,A -85,B 0,C 180,E1 -14465.655,E2 -14465.655} C_VEL
LIN {X 0,Y 340.856,Z 565.472,A -85,B 0,C 180,E1 -14467.257,E2 -14467.257} C_VEL
LIN {X 0,Y 338.922,Z 576.063,A -85,B 0,C 180,E1 -14468.928,E2 -14468.928} C_VEL
LIN {X 0,Y 337.138,Z 586.114,A -85,B 0,C 180,E1 -14470.833,E2 -14470.833} C_VEL
LIN {X 0,Y 335.42,Z 595.403,A -85,B 0,C 180,E1 -14472.943,E2 -14472.943} C_VEL
LIN {X 0,Y 333.92,Z 604.156,A -85,B 0,C 180,E1 -14475.371,E2 -14475.371} C_VEL
LIN {X 0,Y 333.01,Z 611.193,A -85,B 0,C 180,E1 -14477.817,E2 -14477.817} C_VEL
LIN {X 0,Y 332.335,Z 616.728,A -85,B 0,C 180,E1 -14480.26,E2 -14480.26} C_VEL
LIN {X 0,Y 332.049,Z 620.921,A -85,B 0,C 180,E1 -14482.705,E2 -14482.705} C_VEL
LIN {X 0,Y 331.952,Z 623.864,A -85,B 0,C 180,E1 -14485.143,E2 -14485.143} C_VEL
LIN {X 0,Y 331.94,Z 625.619,A -85,B 0,C 180,E1 -14487.574,E2 -14487.574} C_VEL
LIN {X 0,Y 332.042,Z 626.223,A -85,B 0,C 180,E1 -14490.001,E2 -14490.001} C_VEL
LIN {X 0,Y 331.94,Z 625.61,A -85,B 0,C 180,E1 -14492.428,E2 -14492.428} C_VEL
LIN {X 0,Y 331.952,Z 623.844,A -85,B 0,C 180,E1 -14494.859,E2 -14494.859} C_VEL
LIN {X 0,Y 332.045,Z 620.896,A -85,B 0,C 180,E1 -14497.297,E2 -14497.297} C_VEL
LIN {X 0,Y 332.334,Z 616.699,A -85,B 0,C 180,E1 -14499.741,E2 -14499.741} C_VEL
LIN {X 0,Y 333.009,Z 611.151,A -85,B 0,C 180,E1 -14502.184,E2 -14502.184} C_VEL
LIN {X 0,Y 333.921,Z 604.094,A -85,B 0,C 180,E1 -14504.63,E2 -14504.63} C_VEL
LIN {X 0,Y 335.419,Z 595.331,A -85,B 0,C 180,E1 -14507.059,E2 -14507.059} C_VEL
LIN {X 0,Y 337.121,Z 586.03,A -85,B 0,C 180,E1 -14509.169,E2 -14509.169} C_VEL
LIN {X 0,Y 338.922,Z 575.966,A -85,B 0,C 180,E1 -14511.071,E2 -14511.071} C_VEL
LIN {X 0,Y 341.044,Z 564.334,A -85,B 0,C 180,E1 -14512.891,E2 -14512.891} C_VEL
LIN {X 0,Y 343.287,Z 551.856,A -85,B 0,C 180,E1 -14514.493,E2 -14514.493} C_VEL
LIN {X 0,Y 345.542,Z 538.055,A -85,B 0,C 180,E1 -14515.932,E2 -14515.932} C_VEL
LIN {X 0,Y 347.606,Z 523.706,A -85,B 0,C 180,E1 -14517.125,E2 -14517.125} C_VEL
LIN {X 0,Y 349.311,Z 509.454,A -85,B 0,C 180,E1 -14518.054,E2 -14518.054} C_VEL
LIN {X 0,Y 350.831,Z 494.397,A -85,B 0,C 180,E1 -14518.778,E2 -14518.778} C_VEL
LIN {X 0,Y 351.827,Z 480.05,A -85,B 0,C 180,E1 -14519.261,E2 -14519.261} C_VEL
LIN {X 0,Y 354.557,Z 389.767,A -85,B 0,C 180,E1 -14521.117,E2 -14521.117} C_VEL
LIN {X 0,Y 355.294,Z 362.702,A -85,B 0,C 180,E1 -14521.672,E2 -14521.672} C_VEL
LIN {X 0,Y 351.26,Z 339.394,A -85,B 0,C 180,E1 -14522.625,E2 -14522.625} C_VEL
LIN {X 0,Y 350.125,Z 335.533,A -85,B 0,C 180,E1 -14522.834,E2 -14522.834} C_VEL
LIN {X 0,Y 341.069,Z 316.068,A -85,B 0,C 180,E1 -14524.293,E2 -14524.293} C_VEL
LIN {X 0,Y 339.548,Z 312.623,A -85,B 0,C 180,E1 -14524.573,E2 -14524.573} C_VEL
LIN {X 0,Y 336.79,Z 302.401,A -85,B 0,C 180,E1 -14527.241,E2 -14527.241} C_VEL
LIN {X 0,Y 333.662,Z 291.538,A -85,B 0,C 180,E1 -14530.261,E2 -14530.261} C_VEL
LIN {X 0,Y 333.599,Z 291.554,A -85,B 0,C 180,E1 -14534.046,E2 -14534.046} C_VEL
LIN {X 0,Y 333.644,Z 291.543,A -85,B 0,C 180,E1 -14537.619,E2 -14537.619} C_VEL
LIN {X 0,Y 333.655,Z 291.547,A -85,B 0,C 180,E1 -14541.203,E2 -14541.203} C_VEL
LIN {X 0,Y 333.679,Z 291.545,A -85,B 0,C 180,E1 -14543.862,E2 -14543.862} C_VEL
LIN {X 0,Y 333.649,Z 291.541,A -85,B 0,C 180,E1 -14547.413,E2 -14547.413} C_VEL
LIN {X 0,Y 333.659,Z 291.54,A -85,B 0,C 180,E1 -14551.023,E2 -14551.023} C_VEL
LIN {X 0,Y 333.703,Z 291.538,A -85,B 0,C 180,E1 -14555.089,E2 -14555.089} C_VEL
LIN {X 0,Y 333.679,Z 291.544,A -85,B 0,C 180,E1 -14559.019,E2 -14559.019} C_VEL
LIN {X 0,Y 333.798,Z 291.524,A -85,B 0,C 180,E1 -14561.59,E2 -14561.59} C_VEL
LIN {X 0,Y 333.813,Z 291.523,A -85,B 0,C 180,E1 -14565.577,E2 -14565.577} C_VEL
LIN {X 0,Y 333.822,Z 291.519,A -85,B 0,C 180,E1 -14569.078,E2 -14569.078} C_VEL
LIN {X 0,Y 333.961,Z 291.5,A -85,B 0,C 180,E1 -14572.746,E2 -14572.746} C_VEL
LIN {X 0,Y 333.784,Z 291.531,A -85,B 0,C 180,E1 -14575.169,E2 -14575.169} C_VEL
LIN {X 0,Y 334.07,Z 291.489,A -85,B 0,C 180,E1 -14577.589,E2 -14577.589} C_VEL
LIN {X 0,Y 334.064,Z 291.492,A -85,B 0,C 180,E1 -14581.206,E2 -14581.206} C_VEL
LIN {X 0,Y 334.075,Z 291.492,A -85,B 0,C 180,E1 -14582.412,E2 -14582.412} C_VEL
LIN {X 0,Y 333.962,Z 291.501,A -85,B 0,C 180,E1 -14586.478,E2 -14586.478} C_VEL
LIN {X 0,Y 333.824,Z 291.522,A -85,B 0,C 180,E1 -14589.696,E2 -14589.696} C_VEL
LIN {X 0,Y 333.791,Z 291.532,A -85,B 0,C 180,E1 -14593.392,E2 -14593.392} C_VEL
LIN {X 0,Y 333.684,Z 291.545,A -85,B 0,C 180,E1 -14597.15,E2 -14597.15} C_VEL
LIN {X 0,Y 333.648,Z 291.546,A -85,B 0,C 180,E1 -14599.696,E2 -14599.696} C_VEL
LIN {X 0,Y 333.653,Z 291.541,A -85,B 0,C 180,E1 -14602.281,E2 -14602.281} C_VEL
LIN {X 0,Y 333.661,Z 291.548,A -85,B 0,C 180,E1 -14605.078,E2 -14605.078} C_VEL
LIN {X 0,Y 333.632,Z 291.529,A -85,B 0,C 180,E1 -14608.98,E2 -14608.98} C_VEL
LIN {X 0,Y 333.647,Z 291.546,A -85,B 0,C 180,E1 -14612.586,E2 -14612.586} C_VEL
LIN {X 0,Y 333.676,Z 291.54,A -85,B 0,C 180,E1 -14616.139,E2 -14616.139} C_VEL
LIN {X 0,Y 333.604,Z 291.55,A -85,B 0,C 180,E1 -14619.198,E2 -14619.198} C_VEL
LIN {X 0,Y 333.608,Z 291.552,A -85,B 0,C 180,E1 -14622.494,E2 -14622.494} C_VEL
LIN {X 0,Y 333.569,Z 291.555,A -85,B 0,C 180,E1 -14625.949,E2 -14625.949} C_VEL
LIN {X 0,Y 333.597,Z 291.558,A -85,B 0,C 180,E1 -14629.326,E2 -14629.326} C_VEL
LIN {X 0,Y 333.663,Z 291.537,A -85,B 0,C 180,E1 -14633.169,E2 -14633.169} C_VEL
LIN {X 0,Y 333.696,Z 291.625,A -85,B 0,C 180,E1 -14634.646,E2 -14634.646} C_VEL
LIN {X 0,Y 333.845,Z 292.467,A -85,B 0,C 180,E1 -14634.839,E2 -14634.839} C_VEL
LIN {X 0,Y 335.318,Z 295.29,A -85,B 0,C 180,E1 -14635.09,E2 -14635.09} C_VEL
LIN {X 0,Y 342.226,Z 307.667,A -85,B 0,C 180,E1 -14636.21,E2 -14636.21} C_VEL
LIN {X 0,Y 351.541,Z 326.597,A -85,B 0,C 180,E1 -14637.682,E2 -14637.682} C_VEL
LIN {X 0,Y 355.915,Z 336.651,A -85,B 0,C 180,E1 -14638.366,E2 -14638.366} C_VEL
LIN {X 0,Y 353.571,Z 418.758,A -85,B 0,C 180,E1 -14640.039,E2 -14640.039} C_VEL
LIN {X 0,Y 352.373,Z 456.511,A -85,B 0,C 180,E1 -14640.829,E2 -14640.829} C_VEL
LIN {X 0,Y 351.393,Z 472.17,A -85,B 0,C 180,E1 -14641.376,E2 -14641.376} C_VEL
LIN {X 0,Y 350.226,Z 486.754,A -85,B 0,C 180,E1 -14642.124,E2 -14642.124} C_VEL
LIN {X 0,Y 348.735,Z 500.325,A -85,B 0,C 180,E1 -14643.035,E2 -14643.035} C_VEL
LIN {X 0,Y 346.907,Z 513.882,A -85,B 0,C 180,E1 -14644.178,E2 -14644.178} C_VEL
LIN {X 0,Y 344.786,Z 527.631,A -85,B 0,C 180,E1 -14645.62,E2 -14645.62} C_VEL
LIN {X 0,Y 342.793,Z 538.969,A -85,B 0,C 180,E1 -14647.073,E2 -14647.073} C_VEL
LIN {X 0,Y 340.741,Z 550.405,A -85,B 0,C 180,E1 -14648.841,E2 -14648.841} C_VEL
LIN {X 0,Y 338.891,Z 560.025,A -85,B 0,C 180,E1 -14650.621,E2 -14650.621} C_VEL
LIN {X 0,Y 337.047,Z 569.45,A -85,B 0,C 180,E1 -14652.714,E2 -14652.714} C_VEL
LIN {X 0,Y 335.462,Z 577.871,A -85,B 0,C 180,E1 -14654.999,E2 -14654.999} C_VEL
LIN {X 0,Y 334.255,Z 584.601,A -85,B 0,C 180,E1 -14657.245,E2 -14657.245} C_VEL
LIN {X 0,Y 333.298,Z 590.399,A -85,B 0,C 180,E1 -14659.674,E2 -14659.674} C_VEL
LIN {X 0,Y 332.781,Z 593.83,A -85,B 0,C 180,E1 -14661.498,E2 -14661.498} C_VEL
LIN {X 0,Y 332.37,Z 597.301,A -85,B 0,C 180,E1 -14663.93,E2 -14663.93} C_VEL
LIN {X 0,Y 332.128,Z 599.596,A -85,B 0,C 180,E1 -14666.36,E2 -14666.36} C_VEL
LIN {X 0,Y 332.039,Z 600.767,A -85,B 0,C 180,E1 -14668.787,E2 -14668.787} C_VEL
LIN {X 0,Y 332.039,Z 600.782,A -85,B 0,C 180,E1 -14671.212,E2 -14671.212} C_VEL
LIN {X 0,Y 332.127,Z 599.67,A -85,B 0,C 180,E1 -14673.639,E2 -14673.639} C_VEL
LIN {X 0,Y 332.369,Z 597.431,A -85,B 0,C 180,E1 -14676.068,E2 -14676.068} C_VEL
LIN {X 0,Y 332.771,Z 594.012,A -85,B 0,C 180,E1 -14678.501,E2 -14678.501} C_VEL
LIN {X 0,Y 333.45,Z 589.328,A -85,B 0,C 180,E1 -14680.934,E2 -14680.934} C_VEL
LIN {X 0,Y 334.551,Z 583.25,A -85,B 0,C 180,E1 -14683.36,E2 -14683.36} C_VEL
LIN {X 0,Y 335.855,Z 575.597,A -85,B 0,C 180,E1 -14685.785,E2 -14685.785} C_VEL
LIN {X 0,Y 337.497,Z 567.426,A -85,B 0,C 180,E1 -14687.887,E2 -14687.887} C_VEL
LIN {X 0,Y 339.391,Z 557.579,A -85,B 0,C 180,E1 -14689.979,E2 -14689.979} C_VEL
LIN {X 0,Y 341.523,Z 546.494,A -85,B 0,C 180,E1 -14691.913,E2 -14691.913} C_VEL
LIN {X 0,Y 343.61,Z 534.339,A -85,B 0,C 180,E1 -14693.665,E2 -14693.665} C_VEL
LIN {X 0,Y 345.753,Z 522.071,A -85,B 0,C 180,E1 -14695.107,E2 -14695.107} C_VEL
LIN {X 0,Y 347.718,Z 508.657,A -85,B 0,C 180,E1 -14696.401,E2 -14696.401} C_VEL
LIN {X 0,Y 349.378,Z 494.751,A -85,B 0,C 180,E1 -14697.477,E2 -14697.477} C_VEL
LIN {X 0,Y 349.975,Z 489.418,A -85,B 0,C 180,E1 -14697.816,E2 -14697.816} C_VEL
LIN {X 0,Y 349.905,Z 483.976,A -85,B 0,C 180,E1 -14698.197,E2 -14698.197} C_VEL
LIN {X 0,Y 348.115,Z 475.148,A -85,B 0,C 180,E1 -14698.883,E2 -14698.883} C_VEL
LIN {X 0,Y 346.283,Z 466.152,A -85,B 0,C 180,E1 -14699.488,E2 -14699.488} C_VEL
LIN {X 0,Y 346.059,Z 460.459,A -85,B 0,C 180,E1 -14699.733,E2 -14699.733} C_VEL
LIN {X 0,Y 346.873,Z 439.867,A -85,B 0,C 180,E1 -14700.222,E2 -14700.222} C_VEL
LIN {X 0,Y 349.942,Z 340.478,A -85,B 0,C 180,E1 -14702.266,E2 -14702.266} C_VEL
LIN {X 0,Y 349.857,Z 338.634,A -85,B 0,C 180,E1 -14702.319,E2 -14702.319} C_VEL
LIN {X 0,Y 342.075,Z 321.474,A -85,B 0,C 180,E1 -14703.579,E2 -14703.579} C_VEL
LIN {X 0,Y 332.723,Z 303.494,A -85,B 0,C 180,E1 -14705.13,E2 -14705.13} C_VEL
LIN {X 0,Y 328.344,Z 296.21,A -85,B 0,C 180,E1 -14705.868,E2 -14705.868} C_VEL
LIN {X 0,Y 326.949,Z 293.796,A -85,B 0,C 180,E1 -14706.11,E2 -14706.11} C_VEL
LIN {X 0,Y 326.655,Z 292.471,A -85,B 0,C 180,E1 -14706.212,E2 -14706.212} C_VEL
LIN {X 0,Y 326.554,Z 292.432,A -85,B 0,C 180,E1 -14710.214,E2 -14710.214} C_VEL
LIN {X 0,Y 326.557,Z 292.418,A -85,B 0,C 180,E1 -14713.526,E2 -14713.526} C_VEL
LIN {X 0,Y 326.57,Z 292.413,A -85,B 0,C 180,E1 -14717.029,E2 -14717.029} C_VEL
LIN {X 0,Y 326.584,Z 292.431,A -85,B 0,C 180,E1 -14720.778,E2 -14720.778} C_VEL
LIN {X 0,Y 326.608,Z 292.4,A -85,B 0,C 180,E1 -14724.48,E2 -14724.48} C_VEL
LIN {X 0,Y 326.602,Z 292.426,A -85,B 0,C 180,E1 -14727.455,E2 -14727.455} C_VEL
LIN {X 0,Y 326.576,Z 292.43,A -85,B 0,C 180,E1 -14730.332,E2 -14730.332} C_VEL
LIN {X 0,Y 326.593,Z 292.423,A -85,B 0,C 180,E1 -14733.134,E2 -14733.134} C_VEL
LIN {X 0,Y 326.588,Z 292.421,A -85,B 0,C 180,E1 -14737.21,E2 -14737.21} C_VEL
LIN {X 0,Y 326.645,Z 292.41,A -85,B 0,C 180,E1 -14741.206,E2 -14741.206} C_VEL
LIN {X 0,Y 326.723,Z 292.402,A -85,B 0,C 180,E1 -14745.459,E2 -14745.459} C_VEL
LIN {X 0,Y 326.755,Z 292.406,A -85,B 0,C 180,E1 -14748.838,E2 -14748.838} C_VEL
LIN {X 0,Y 326.91,Z 292.388,A -85,B 0,C 180,E1 -14752.589,E2 -14752.589} C_VEL
LIN {X 0,Y 326.752,Z 292.4,A -85,B 0,C 180,E1 -14755.064,E2 -14755.064} C_VEL
LIN {X 0,Y 327.031,Z 292.369,A -85,B 0,C 180,E1 -14757.536,E2 -14757.536} C_VEL
LIN {X 0,Y 327.044,Z 292.358,A -85,B 0,C 180,E1 -14761.231,E2 -14761.231} C_VEL
LIN {X 0,Y 326.758,Z 292.408,A -85,B 0,C 180,E1 -14763.699,E2 -14763.699} C_VEL
LIN {X 0,Y 326.942,Z 292.374,A -85,B 0,C 180,E1 -14766.17,E2 -14766.17} C_VEL
LIN {X 0,Y 326.781,Z 292.398,A -85,B 0,C 180,E1 -14769.907,E2 -14769.907} C_VEL
LIN {X 0,Y 326.758,Z 292.409,A -85,B 0,C 180,E1 -14773.685,E2 -14773.685} C_VEL
LIN {X 0,Y 326.698,Z 292.417,A -85,B 0,C 180,E1 -14777.528,E2 -14777.528} C_VEL
LIN {X 0,Y 326.661,Z 292.415,A -85,B 0,C 180,E1 -14780.135,E2 -14780.135} C_VEL
LIN {X 0,Y 326.616,Z 292.421,A -85,B 0,C 180,E1 -14782.788,E2 -14782.788} C_VEL
LIN {X 0,Y 326.634,Z 292.391,A -85,B 0,C 180,E1 -14785.488,E2 -14785.488} C_VEL
LIN {X 0,Y 326.619,Z 292.426,A -85,B 0,C 180,E1 -14788.254,E2 -14788.254} C_VEL
LIN {X 0,Y 326.571,Z 292.409,A -85,B 0,C 180,E1 -14791.097,E2 -14791.097} C_VEL
LIN {X 0,Y 326.606,Z 292.421,A -85,B 0,C 180,E1 -14794.019,E2 -14794.019} C_VEL
LIN {X 0,Y 326.626,Z 292.404,A -85,B 0,C 180,E1 -14797.239,E2 -14797.239} C_VEL
LIN {X 0,Y 326.576,Z 292.428,A -85,B 0,C 180,E1 -14801.132,E2 -14801.132} C_VEL
LIN {X 0,Y 326.525,Z 292.434,A -85,B 0,C 180,E1 -14804.743,E2 -14804.743} C_VEL
LIN {X 0,Y 326.574,Z 292.425,A -85,B 0,C 180,E1 -14808.155,E2 -14808.155} C_VEL
LIN {X 0,Y 326.59,Z 292.425,A -85,B 0,C 180,E1 -14808.97,E2 -14808.97} C_VEL
LIN {X 0,Y 329.765,Z 303.127,A -85,B 0,C 180,E1 -14812.05,E2 -14812.05} C_VEL
LIN {X 0,Y 332.338,Z 312.578,A -85,B 0,C 180,E1 -14814.567,E2 -14814.567} C_VEL
LIN {X 0,Y 341.989,Z 332.872,A -85,B 0,C 180,E1 -14816.202,E2 -14816.202} C_VEL
LIN {X 0,Y 345.314,Z 340.717,A -85,B 0,C 180,E1 -14816.758,E2 -14816.758} C_VEL
LIN {X 0,Y 348.59,Z 359.607,A -85,B 0,C 180,E1 -14817.558,E2 -14817.558} C_VEL
LIN {X 0,Y 349.349,Z 364.449,A -85,B 0,C 180,E1 -14817.752,E2 -14817.752} C_VEL
LIN {X 0,Y 345.737,Z 479.119,A -85,B 0,C 180,E1 -14820.131,E2 -14820.131} C_VEL
LIN {X 0,Y 344.639,Z 494.571,A -85,B 0,C 180,E1 -14820.656,E2 -14820.656} C_VEL
LIN {X 0,Y 343.071,Z 509.499,A -85,B 0,C 180,E1 -14821.39,E2 -14821.39} C_VEL
LIN {X 0,Y 341.188,Z 524.447,A -85,B 0,C 180,E1 -14822.386,E2 -14822.386} C_VEL
LIN {X 0,Y 339.136,Z 537.981,A -85,B 0,C 180,E1 -14823.542,E2 -14823.542} C_VEL
LIN {X 0,Y 336.783,Z 551.73,A -85,B 0,C 180,E1 -14825.003,E2 -14825.003} C_VEL
LIN {X 0,Y 334.462,Z 564.184,A -85,B 0,C 180,E1 -14826.634,E2 -14826.634} C_VEL
LIN {X 0,Y 332.11,Z 576.499,A -85,B 0,C 180,E1 -14828.609,E2 -14828.609} C_VEL
LIN {X 0,Y 330.08,Z 587.287,A -85,B 0,C 180,E1 -14830.73,E2 -14830.73} C_VEL
LIN {X 0,Y 328.321,Z 596.354,A -85,B 0,C 180,E1 -14832.883,E2 -14832.883} C_VEL
LIN {X 0,Y 326.986,Z 603.884,A -85,B 0,C 180,E1 -14835.054,E2 -14835.054} C_VEL
LIN {X 0,Y 326.005,Z 610.921,A -85,B 0,C 180,E1 -14837.551,E2 -14837.551} C_VEL
LIN {X 0,Y 325.293,Z 616.457,A -85,B 0,C 180,E1 -14840.048,E2 -14840.048} C_VEL
LIN {X 0,Y 324.968,Z 620.65,A -85,B 0,C 180,E1 -14842.545,E2 -14842.545} C_VEL
LIN {X 0,Y 324.864,Z 623.593,A -85,B 0,C 180,E1 -14845.036,E2 -14845.036} C_VEL
LIN {X 0,Y 324.858,Z 625.349,A -85,B 0,C 180,E1 -14847.521,E2 -14847.521} C_VEL
LIN {X 0,Y 324.946,Z 625.952,A -85,B 0,C 180,E1 -14850.001,E2 -14850.001} C_VEL
LIN {X 0,Y 324.858,Z 625.34,A -85,B 0,C 180,E1 -14852.48,E2 -14852.48} C_VEL
LIN {X 0,Y 324.864,Z 623.573,A -85,B 0,C 180,E1 -14854.965,E2 -14854.965} C_VEL
LIN {X 0,Y 324.965,Z 620.623,A -85,B 0,C 180,E1 -14857.456,E2 -14857.456} C_VEL
LIN {X 0,Y 325.292,Z 616.426,A -85,B 0,C 180,E1 -14859.954,E2 -14859.954} C_VEL
LIN {X 0,Y 326.005,Z 610.876,A -85,B 0,C 180,E1 -14862.45,E2 -14862.45} C_VEL
LIN {X 0,Y 326.986,Z 603.819,A -85,B 0,C 180,E1 -14864.947,E2 -14864.947} C_VEL
LIN {X 0,Y 328.54,Z 595.055,A -85,B 0,C 180,E1 -14867.427,E2 -14867.427} C_VEL
LIN {X 0,Y 330.352,Z 585.755,A -85,B 0,C 180,E1 -14869.577,E2 -14869.577} C_VEL
LIN {X 0,Y 332.124,Z 576.368,A -85,B 0,C 180,E1 -14871.397,E2 -14871.397} C_VEL
LIN {X 0,Y 334.262,Z 565.088,A -85,B 0,C 180,E1 -14873.218,E2 -14873.218} C_VEL
LIN {X 0,Y 336.569,Z 552.808,A -85,B 0,C 180,E1 -14874.85,E2 -14874.85} C_VEL
LIN {X 0,Y 338.897,Z 539.312,A -85,B 0,C 180,E1 -14876.314,E2 -14876.314} C_VEL
LIN {X 0,Y 341.146,Z 524.503,A -85,B 0,C 180,E1 -14877.592,E2 -14877.592} C_VEL
LIN {X 0,Y 342.909,Z 510.43,A -85,B 0,C 180,E1 -14878.542,E2 -14878.542} C_VEL
LIN {X 0,Y 344.542,Z 495.008,A -85,B 0,C 180,E1 -14879.312,E2 -14879.312} C_VEL
LIN {X 0,Y 345.652,Z 479.766,A -85,B 0,C 180,E1 -14879.836,E2 -14879.836} C_VEL
LIN {X 0,Y 348.493,Z 389.476,A -85,B 0,C 180,E1 -14881.721,E2 -14881.721} C_VEL
LIN {X 0,Y 349.234,Z 363.669,A -85,B 0,C 180,E1 -14882.257,E2 -14882.257} C_VEL
LIN {X 0,Y 345.115,Z 339.989,A -85,B 0,C 180,E1 -14883.258,E2 -14883.258} C_VEL
LIN {X 0,Y 336.041,Z 320.215,A -85,B 0,C 180,E1 -14884.768,E2 -14884.768} C_VEL
LIN {X 0,Y 332.247,Z 312.222,A -85,B 0,C 180,E1 -14885.462,E2 -14885.462} C_VEL
LIN {X 0,Y 329.064,Z 300.717,A -85,B 0,C 180,E1 -14888.595,E2 -14888.595} C_VEL
LIN {X 0,Y 326.594,Z 292.429,A -85,B 0,C 180,E1 -14891.031,E2 -14891.031} C_VEL
LIN {X 0,Y 326.53,Z 292.437,A -85,B 0,C 180,E1 -14894.743,E2 -14894.743} C_VEL
LIN {X 0,Y 326.579,Z 292.428,A -85,B 0,C 180,E1 -14898.155,E2 -14898.155} C_VEL
LIN {X 0,Y 326.626,Z 292.423,A -85,B 0,C 180,E1 -14901.392,E2 -14901.392} C_VEL
LIN {X 0,Y 326.622,Z 292.418,A -85,B 0,C 180,E1 -14904.852,E2 -14904.852} C_VEL
LIN {X 0,Y 326.613,Z 292.417,A -85,B 0,C 180,E1 -14907.456,E2 -14907.456} C_VEL
LIN {X 0,Y 326.621,Z 292.416,A -85,B 0,C 180,E1 -14910.337,E2 -14910.337} C_VEL
LIN {X 0,Y 326.647,Z 292.417,A -85,B 0,C 180,E1 -14914.644,E2 -14914.644} C_VEL
LIN {X 0,Y 326.625,Z 292.424,A -85,B 0,C 180,E1 -14918.544,E2 -14918.544} C_VEL
LIN {X 0,Y 326.749,Z 292.4,A -85,B 0,C 180,E1 -14921.178,E2 -14921.178} C_VEL
LIN {X 0,Y 326.768,Z 292.399,A -85,B 0,C 180,E1 -14925.433,E2 -14925.433} C_VEL
LIN {X 0,Y 326.763,Z 292.398,A -85,B 0,C 180,E1 -14928.839,E2 -14928.839} C_VEL
LIN {X 0,Y 326.918,Z 292.378,A -85,B 0,C 180,E1 -14932.589,E2 -14932.589} C_VEL
LIN {X 0,Y 326.753,Z 292.407,A -85,B 0,C 180,E1 -14935.065,E2 -14935.065} C_VEL
LIN {X 0,Y 327.014,Z 292.367,A -85,B 0,C 180,E1 -14937.537,E2 -14937.537} C_VEL
LIN {X 0,Y 327.034,Z 292.367,A -85,B 0,C 180,E1 -14941.232,E2 -14941.232} C_VEL
LIN {X 0,Y 326.766,Z 292.408,A -85,B 0,C 180,E1 -14943.7,E2 -14943.7} C_VEL
LIN {X 0,Y 326.924,Z 292.378,A -85,B 0,C 180,E1 -14946.466,E2 -14946.466} C_VEL
LIN {X 0,Y 326.787,Z 292.396,A -85,B 0,C 180,E1 -14949.907,E2 -14949.907} C_VEL
LIN {X 0,Y 326.747,Z 292.405,A -85,B 0,C 180,E1 -14953.686,E2 -14953.686} C_VEL
LIN {X 0,Y 326.632,Z 292.422,A -85,B 0,C 180,E1 -14957.532,E2 -14957.532} C_VEL
LIN {X 0,Y 326.611,Z 292.426,A -85,B 0,C 180,E1 -14961.457,E2 -14961.457} C_VEL
LIN {X 0,Y 326.604,Z 292.424,A -85,B 0,C 180,E1 -14965.491,E2 -14965.491} C_VEL
LIN {X 0,Y 326.593,Z 292.4,A -85,B 0,C 180,E1 -14968.257,E2 -14968.257} C_VEL
LIN {X 0,Y 326.576,Z 292.43,A -85,B 0,C 180,E1 -14971.097,E2 -14971.097} C_VEL
LIN {X 0,Y 326.61,Z 292.426,A -85,B 0,C 180,E1 -14974.019,E2 -14974.019} C_VEL
LIN {X 0,Y 326.625,Z 292.424,A -85,B 0,C 180,E1 -14977.237,E2 -14977.237} C_VEL
LIN {X 0,Y 326.536,Z 292.431,A -85,B 0,C 180,E1 -14981.122,E2 -14981.122} C_VEL
LIN {X 0,Y 326.513,Z 292.436,A -85,B 0,C 180,E1 -14984.739,E2 -14984.739} C_VEL
LIN {X 0,Y 326.536,Z 292.431,A -85,B 0,C 180,E1 -14988.147,E2 -14988.147} C_VEL
LIN {X 0,Y 326.584,Z 292.43,A -85,B 0,C 180,E1 -14991.385,E2 -14991.385} C_VEL
LIN {X 0,Y 326.661,Z 292.469,A -85,B 0,C 180,E1 -14993.909,E2 -14993.909} C_VEL
LIN {X 0,Y 327.764,Z 295.488,A -85,B 0,C 180,E1 -14994.159,E2 -14994.159} C_VEL
LIN {X 0,Y 329.405,Z 297.93,A -85,B 0,C 180,E1 -14994.431,E2 -14994.431} C_VEL
LIN {X 0,Y 336.713,Z 310.858,A -85,B 0,C 180,E1 -14995.654,E2 -14995.654} C_VEL
LIN {X 0,Y 345.741,Z 329.276,A -85,B 0,C 180,E1 -14997.13,E2 -14997.13} C_VEL
LIN {X 0,Y 349.835,Z 338.676,A -85,B 0,C 180,E1 -14997.791,E2 -14997.791} C_VEL
LIN {X 0,Y 347.501,Z 417.975,A -85,B 0,C 180,E1 -14999.435,E2 -14999.435} C_VEL
LIN {X 0,Y 346.217,Z 456.798,A -85,B 0,C 180,E1 -15000.259,E2 -15000.259} C_VEL
LIN {X 0,Y 345.183,Z 472.511,A -85,B 0,C 180,E1 -15000.815,E2 -15000.815} C_VEL
LIN {X 0,Y 343.997,Z 486.871,A -85,B 0,C 180,E1 -15001.563,E2 -15001.563} C_VEL
LIN {X 0,Y 342.434,Z 500.602,A -85,B 0,C 180,E1 -15002.497,E2 -15002.497} C_VEL
LIN {X 0,Y 340.522,Z 514.158,A -85,B 0,C 180,E1 -15003.657,E2 -15003.657} C_VEL
LIN {X 0,Y 338.34,Z 527.906,A -85,B 0,C 180,E1 -15005.125,E2 -15005.125} C_VEL
LIN {X 0,Y 336.247,Z 539.244,A -85,B 0,C 180,E1 -15006.601,E2 -15006.601} C_VEL
LIN {X 0,Y 334.133,Z 550.679,A -85,B 0,C 180,E1 -15008.402,E2 -15008.402} C_VEL
LIN {X 0,Y 332.178,Z 560.299,A -85,B 0,C 180,E1 -15010.213,E2 -15010.213} C_VEL
LIN {X 0,Y 330.234,Z 569.724,A -85,B 0,C 180,E1 -15012.345,E2 -15012.345} C_VEL
LIN {X 0,Y 328.534,Z 578.33,A -85,B 0,C 180,E1 -15014.735,E2 -15014.735} C_VEL
LIN {X 0,Y 327.302,Z 584.874,A -85,B 0,C 180,E1 -15016.969,E2 -15016.969} C_VEL
LIN {X 0,Y 326.277,Z 590.672,A -85,B 0,C 180,E1 -15019.45,E2 -15019.45} C_VEL
LIN {X 0,Y 325.745,Z 594.102,A -85,B 0,C 180,E1 -15021.313,E2 -15021.313} C_VEL
LIN {X 0,Y 325.321,Z 597.572,A -85,B 0,C 180,E1 -15023.798,E2 -15023.798} C_VEL
LIN {X 0,Y 325.058,Z 599.867,A -85,B 0,C 180,E1 -15026.28,E2 -15026.28} C_VEL
LIN {X 0,Y 324.945,Z 601.037,A -85,B 0,C 180,E1 -15028.76,E2 -15028.76} C_VEL
LIN {X 0,Y 324.945,Z 601.052,A -85,B 0,C 180,E1 -15031.239,E2 -15031.239} C_VEL
LIN {X 0,Y 325.057,Z 599.939,A -85,B 0,C 180,E1 -15033.718,E2 -15033.718} C_VEL
LIN {X 0,Y 325.367,Z 597.379,A -85,B 0,C 180,E1 -15036.479,E2 -15036.479} C_VEL
LIN {X 0,Y 325.91,Z 593.231,A -85,B 0,C 180,E1 -15039.307,E2 -15039.307} C_VEL
LIN {X 0,Y 326.681,Z 588.194,A -85,B 0,C 180,E1 -15041.792,E2 -15041.792} C_VEL
LIN {X 0,Y 327.94,Z 581.732,A -85,B 0,C 180,E1 -15044.267,E2 -15044.267} C_VEL
LIN {X 0,Y 329.224,Z 574.761,A -85,B 0,C 180,E1 -15046.43,E2 -15046.43} C_VEL
LIN {X 0,Y 330.961,Z 566.361,A -85,B 0,C 180,E1 -15048.573,E2 -15048.573} C_VEL
LIN {X 0,Y 333.021,Z 556.24,A -85,B 0,C 180,E1 -15050.7,E2 -15050.7} C_VEL
LIN {X 0,Y 335.013,Z 546.217,A -85,B 0,C 180,E1 -15052.453,E2 -15052.453} C_VEL
LIN {X 0,Y 337.102,Z 534.606,A -85,B 0,C 180,E1 -15054.151,E2 -15054.151} C_VEL
LIN {X 0,Y 339.328,Z 522.337,A -85,B 0,C 180,E1 -15055.616,E2 -15055.616} C_VEL
LIN {X 0,Y 341.369,Z 508.922,A -85,B 0,C 180,E1 -15056.931,E2 -15056.931} C_VEL
LIN {X 0,Y 343.103,Z 495.014,A -85,B 0,C 180,E1 -15058.024,E2 -15058.024} C_VEL
LIN {X 0,Y 344.633,Z 479.883,A -85,B 0,C 180,E1 -15058.939,E2 -15058.939} C_VEL
LIN {X 0,Y 345.847,Z 464.389,A -85,B 0,C 180,E1 -15059.607,E2 -15059.607} C_VEL
LIN {X 0,Y 346.059,Z 460.459,A -85,B 0,C 180,E1 -15059.733,E2 -15059.733} C_VEL
LIN {X 0,Y 345.829,Z 454.704,A -85,B 0,C 180,E1 -15059.953,E2 -15059.953} C_VEL
LIN {X 0,Y 341.438,Z 436.106,A -85,B 0,C 180,E1 -15060.855,E2 -15060.855} C_VEL
LIN {X 0,Y 341.033,Z 430.3,A -85,B 0,C 180,E1 -15061.031,E2 -15061.031} C_VEL
LIN {X 0,Y 343.961,Z 341.255,A -85,B 0,C 180,E1 -15062.885,E2 -15062.885} C_VEL
LIN {X 0,Y 339.794,Z 331.558,A -85,B 0,C 180,E1 -15063.586,E2 -15063.586} C_VEL
LIN {X 0,Y 331.173,Z 314.024,A -85,B 0,C 180,E1 -15065.046,E2 -15065.046} C_VEL
LIN {X 0,Y 325.768,Z 304.335,A -85,B 0,C 180,E1 -15065.981,E2 -15065.981} C_VEL
LIN {X 0,Y 321.458,Z 297.296,A -85,B 0,C 180,E1 -15066.738,E2 -15066.738} C_VEL
LIN {X 0,Y 320.037,Z 295.003,A -85,B 0,C 180,E1 -15066.993,E2 -15066.993} C_VEL
LIN {X 0,Y 319.591,Z 293.301,A -85,B 0,C 180,E1 -15067.136,E2 -15067.136} C_VEL
LIN {X 0,Y 319.527,Z 293.309,A -85,B 0,C 180,E1 -15069.661,E2 -15069.661} C_VEL
LIN {X 0,Y 319.516,Z 293.294,A -85,B 0,C 180,E1 -15073.459,E2 -15073.459} C_VEL
LIN {X 0,Y 319.548,Z 293.287,A -85,B 0,C 180,E1 -15077.015,E2 -15077.015} C_VEL
LIN {X 0,Y 319.528,Z 293.308,A -85,B 0,C 180,E1 -15080.368,E2 -15080.368} C_VEL
LIN {X 0,Y 319.575,Z 293.275,A -85,B 0,C 180,E1 -15084.457,E2 -15084.457} C_VEL
LIN {X 0,Y 319.517,Z 293.306,A -85,B 0,C 180,E1 -15088.136,E2 -15088.136} C_VEL
LIN {X 0,Y 319.541,Z 293.304,A -85,B 0,C 180,E1 -15091.613,E2 -15091.613} C_VEL
LIN {X 0,Y 319.536,Z 293.305,A -85,B 0,C 180,E1 -15095.298,E2 -15095.298} C_VEL
LIN {X 0,Y 319.56,Z 293.3,A -85,B 0,C 180,E1 -15098.045,E2 -15098.045} C_VEL
LIN {X 0,Y 319.581,Z 293.293,A -85,B 0,C 180,E1 -15102.068,E2 -15102.068} C_VEL
LIN {X 0,Y 319.707,Z 293.275,A -85,B 0,C 180,E1 -15106.007,E2 -15106.007} C_VEL
LIN {X 0,Y 319.733,Z 293.277,A -85,B 0,C 180,E1 -15109.872,E2 -15109.872} C_VEL
LIN {X 0,Y 319.895,Z 293.262,A -85,B 0,C 180,E1 -15113.693,E2 -15113.693} C_VEL
LIN {X 0,Y 319.974,Z 293.248,A -85,B 0,C 180,E1 -15117.482,E2 -15117.482} C_VEL
LIN {X 0,Y 320.012,Z 293.234,A -85,B 0,C 180,E1 -15121.258,E2 -15121.258} C_VEL
LIN {X 0,Y 319.721,Z 293.277,A -85,B 0,C 180,E1 -15125.044,E2 -15125.044} C_VEL
LIN {X 0,Y 319.851,Z 293.264,A -85,B 0,C 180,E1 -15127.576,E2 -15127.576} C_VEL
LIN {X 0,Y 319.713,Z 293.276,A -85,B 0,C 180,E1 -15131.411,E2 -15131.411} C_VEL
LIN {X 0,Y 319.698,Z 293.277,A -85,B 0,C 180,E1 -15135.295,E2 -15135.295} C_VEL
LIN {X 0,Y 319.672,Z 293.283,A -85,B 0,C 180,E1 -15139.255,E2 -15139.255} C_VEL
LIN {X 0,Y 319.562,Z 293.29,A -85,B 0,C 180,E1 -15143.32,E2 -15143.32} C_VEL
LIN {X 0,Y 319.569,Z 293.274,A -85,B 0,C 180,E1 -15146.094,E2 -15146.094} C_VEL
LIN {X 0,Y 319.55,Z 293.305,A -85,B 0,C 180,E1 -15148.937,E2 -15148.937} C_VEL
LIN {X 0,Y 319.523,Z 293.282,A -85,B 0,C 180,E1 -15151.863,E2 -15151.863} C_VEL
LIN {X 0,Y 319.578,Z 293.299,A -85,B 0,C 180,E1 -15155.543,E2 -15155.543} C_VEL
LIN {X 0,Y 319.556,Z 293.305,A -85,B 0,C 180,E1 -15159.669,E2 -15159.669} C_VEL
LIN {X 0,Y 319.52,Z 293.307,A -85,B 0,C 180,E1 -15163.461,E2 -15163.461} C_VEL
LIN {X 0,Y 319.519,Z 293.308,A -85,B 0,C 180,E1 -15167.763,E2 -15167.763} C_VEL
LIN {X 0,Y 319.557,Z 293.422,A -85,B 0,C 180,E1 -15168.212,E2 -15168.212} C_VEL
LIN {X 0,Y 322.958,Z 304.702,A -85,B 0,C 180,E1 -15171.574,E2 -15171.574} C_VEL
LIN {X 0,Y 325.089,Z 312.36,A -85,B 0,C 180,E1 -15173.656,E2 -15173.656} C_VEL
LIN {X 0,Y 333.803,Z 330.198,A -85,B 0,C 180,E1 -15175.197,E2 -15175.197} C_VEL
LIN {X 0,Y 339.625,Z 343.36,A -85,B 0,C 180,E1 -15176.198,E2 -15176.198} C_VEL
LIN {X 0,Y 343.261,Z 364.738,A -85,B 0,C 180,E1 -15177.122,E2 -15177.122} C_VEL
LIN {X 0,Y 340.325,Z 458.722,A -85,B 0,C 180,E1 -15179.091,E2 -15179.091} C_VEL
LIN {X 0,Y 339.438,Z 481.254,A -85,B 0,C 180,E1 -15179.605,E2 -15179.605} C_VEL
LIN {X 0,Y 338.228,Z 496.677,A -85,B 0,C 180,E1 -15180.173,E2 -15180.173} C_VEL
LIN {X 0,Y 336.534,Z 511.582,A -85,B 0,C 180,E1 -15180.953,E2 -15180.953} C_VEL
LIN {X 0,Y 334.751,Z 525.101,A -85,B 0,C 180,E1 -15181.893,E2 -15181.893} C_VEL
LIN {X 0,Y 332.519,Z 539.226,A -85,B 0,C 180,E1 -15183.143,E2 -15183.143} C_VEL
LIN {X 0,Y 330.081,Z 552.675,A -85,B 0,C 180,E1 -15184.628,E2 -15184.628} C_VEL
LIN {X 0,Y 327.687,Z 564.932,A -85,B 0,C 180,E1 -15186.289,E2 -15186.289} C_VEL
LIN {X 0,Y 325.428,Z 576.302,A -85,B 0,C 180,E1 -15188.162,E2 -15188.162} C_VEL
LIN {X 0,Y 323.327,Z 587.016,A -85,B 0,C 180,E1 -15190.311,E2 -15190.311} C_VEL
LIN {X 0,Y 321.475,Z 596.082,A -85,B 0,C 180,E1 -15192.507,E2 -15192.507} C_VEL
LIN {X 0,Y 320.058,Z 603.612,A -85,B 0,C 180,E1 -15194.723,E2 -15194.723} C_VEL
LIN {X 0,Y 318.991,Z 610.648,A -85,B 0,C 180,E1 -15197.273,E2 -15197.273} C_VEL
LIN {X 0,Y 318.243,Z 616.185,A -85,B 0,C 180,E1 -15199.825,E2 -15199.825} C_VEL
LIN {X 0,Y 317.886,Z 620.378,A -85,B 0,C 180,E1 -15202.378,E2 -15202.378} C_VEL
LIN {X 0,Y 317.78,Z 623.323,A -85,B 0,C 180,E1 -15204.925,E2 -15204.925} C_VEL
LIN {X 0,Y 317.777,Z 625.079,A -85,B 0,C 180,E1 -15207.465,E2 -15207.465} C_VEL
LIN {X 0,Y 317.851,Z 625.682,A -85,B 0,C 180,E1 -15210.001,E2 -15210.001} C_VEL
LIN {X 0,Y 317.777,Z 625.07,A -85,B 0,C 180,E1 -15212.536,E2 -15212.536} C_VEL
LIN {X 0,Y 317.78,Z 623.301,A -85,B 0,C 180,E1 -15215.076,E2 -15215.076} C_VEL
LIN {X 0,Y 317.884,Z 620.35,A -85,B 0,C 180,E1 -15217.624,E2 -15217.624} C_VEL
LIN {X 0,Y 318.235,Z 616.152,A -85,B 0,C 180,E1 -15220.177,E2 -15220.177} C_VEL
LIN {X 0,Y 318.992,Z 610.601,A -85,B 0,C 180,E1 -15222.728,E2 -15222.728} C_VEL
LIN {X 0,Y 320.059,Z 603.545,A -85,B 0,C 180,E1 -15225.279,E2 -15225.279} C_VEL
LIN {X 0,Y 321.695,Z 594.779,A -85,B 0,C 180,E1 -15227.81,E2 -15227.81} C_VEL
LIN {X 0,Y 323.311,Z 586.932,A -85,B 0,C 180,E1 -15229.691,E2 -15229.691} C_VEL
LIN {X 0,Y 325.431,Z 576.198,A -85,B 0,C 180,E1 -15231.839,E2 -15231.839} C_VEL
LIN {X 0,Y 327.683,Z 564.812,A -85,B 0,C 180,E1 -15233.713,E2 -15233.713} C_VEL
LIN {X 0,Y 330.074,Z 552.532,A -85,B 0,C 180,E1 -15235.373,E2 -15235.373} C_VEL
LIN {X 0,Y 332.528,Z 539.036,A -85,B 0,C 180,E1 -15236.858,E2 -15236.858} C_VEL
LIN {X 0,Y 334.697,Z 525.187,A -85,B 0,C 180,E1 -15238.081,E2 -15238.081} C_VEL
LIN {X 0,Y 336.663,Z 510.151,A -85,B 0,C 180,E1 -15239.122,E2 -15239.122} C_VEL
LIN {X 0,Y 338.374,Z 494.728,A -85,B 0,C 180,E1 -15239.9,E2 -15239.9} C_VEL
LIN {X 0,Y 339.513,Z 479.481,A -85,B 0,C 180,E1 -15240.432,E2 -15240.432} C_VEL
LIN {X 0,Y 342.448,Z 389.941,A -85,B 0,C 180,E1 -15242.33,E2 -15242.33} C_VEL
LIN {X 0,Y 343.201,Z 364.827,A -85,B 0,C 180,E1 -15242.86,E2 -15242.86} C_VEL
LIN {X 0,Y 339.416,Z 342.767,A -85,B 0,C 180,E1 -15243.816,E2 -15243.816} C_VEL
LIN {X 0,Y 330.672,Z 323.684,A -85,B 0,C 180,E1 -15245.32,E2 -15245.32} C_VEL
LIN {X 0,Y 324.944,Z 311.915,A -85,B 0,C 180,E1 -15246.377,E2 -15246.377} C_VEL
LIN {X 0,Y 321.673,Z 300.324,A -85,B 0,C 180,E1 -15249.666,E2 -15249.666} C_VEL
LIN {X 0,Y 319.536,Z 293.305,A -85,B 0,C 180,E1 -15251.818,E2 -15251.818} C_VEL
LIN {X 0,Y 319.49,Z 293.307,A -85,B 0,C 180,E1 -15255.258,E2 -15255.258} C_VEL
LIN {X 0,Y 319.532,Z 293.309,A -85,B 0,C 180,E1 -15258.712,E2 -15258.712} C_VEL
LIN {X 0,Y 319.564,Z 293.299,A -85,B 0,C 180,E1 -15262.348,E2 -15262.348} C_VEL
LIN {X 0,Y 319.563,Z 293.297,A -85,B 0,C 180,E1 -15265.124,E2 -15265.124} C_VEL
LIN {X 0,Y 319.529,Z 293.301,A -85,B 0,C 180,E1 -15268.138,E2 -15268.138} C_VEL
LIN {X 0,Y 319.576,Z 293.296,A -85,B 0,C 180,E1 -15271.604,E2 -15271.604} C_VEL
LIN {X 0,Y 319.579,Z 293.298,A -85,B 0,C 180,E1 -15275.302,E2 -15275.302} C_VEL
LIN {X 0,Y 319.607,Z 293.297,A -85,B 0,C 180,E1 -15279.401,E2 -15279.401} C_VEL
LIN {X 0,Y 319.663,Z 293.289,A -85,B 0,C 180,E1 -15282.074,E2 -15282.074} C_VEL
LIN {X 0,Y 319.737,Z 293.28,A -85,B 0,C 180,E1 -15286.008,E2 -15286.008} C_VEL
LIN {X 0,Y 319.74,Z 293.278,A -85,B 0,C 180,E1 -15289.872,E2 -15289.872} C_VEL
LIN {X 0,Y 319.904,Z 293.254,A -85,B 0,C 180,E1 -15293.694,E2 -15293.694} C_VEL
LIN {X 0,Y 319.96,Z 293.245,A -85,B 0,C 180,E1 -15297.482,E2 -15297.482} C_VEL
LIN {X 0,Y 320.003,Z 293.242,A -85,B 0,C 180,E1 -15301.259,E2 -15301.259} C_VEL
LIN {X 0,Y 319.716,Z 293.287,A -85,B 0,C 180,E1 -15303.781,E2 -15303.781} C_VEL
LIN {X 0,Y 319.889,Z 293.255,A -85,B 0,C 180,E1 -15306.448,E2 -15306.448} C_VEL
LIN {X 0,Y 319.739,Z 293.273,A -85,B 0,C 180,E1 -15310.128,E2 -15310.128} C_VEL
LIN {X 0,Y 319.714,Z 293.278,A -85,B 0,C 180,E1 -15313.993,E2 -15313.993} C_VEL
LIN {X 0,Y 319.588,Z 293.295,A -85,B 0,C 180,E1 -15317.931,E2 -15317.931} C_VEL
LIN {X 0,Y 319.566,Z 293.298,A -85,B 0,C 180,E1 -15321.955,E2 -15321.955} C_VEL
LIN {X 0,Y 319.553,Z 293.296,A -85,B 0,C 180,E1 -15326.095,E2 -15326.095} C_VEL
LIN {X 0,Y 319.527,Z 293.284,A -85,B 0,C 180,E1 -15328.94,E2 -15328.94} C_VEL
LIN {X 0,Y 319.527,Z 293.307,A -85,B 0,C 180,E1 -15331.862,E2 -15331.862} C_VEL
LIN {X 0,Y 319.581,Z 293.297,A -85,B 0,C 180,E1 -15335.542,E2 -15335.542} C_VEL
LIN {X 0,Y 319.531,Z 293.306,A -85,B 0,C 180,E1 -15339.662,E2 -15339.662} C_VEL
LIN {X 0,Y 319.486,Z 293.309,A -85,B 0,C 180,E1 -15343.453,E2 -15343.453} C_VEL
LIN {X 0,Y 319.472,Z 293.314,A -85,B 0,C 180,E1 -15347.002,E2 -15347.002} C_VEL
LIN {X 0,Y 319.517,Z 293.307,A -85,B 0,C 180,E1 -15350.366,E2 -15350.366} C_VEL
LIN {X 0,Y 319.59,Z 293.289,A -85,B 0,C 180,E1 -15353.007,E2 -15353.007} C_VEL
LIN {X 0,Y 320.718,Z 296.337,A -85,B 0,C 180,E1 -15353.257,E2 -15353.257} C_VEL
LIN {X 0,Y 322.185,Z 298.399,A -85,B 0,C 180,E1 -15353.51,E2 -15353.51} C_VEL
LIN {X 0,Y 328.798,Z 309.596,A -85,B 0,C 180,E1 -15354.662,E2 -15354.662} C_VEL
LIN {X 0,Y 337.63,Z 326.953,A -85,B 0,C 180,E1 -15356.167,E2 -15356.167} C_VEL
LIN {X 0,Y 343.835,Z 340.763,A -85,B 0,C 180,E1 -15357.203,E2 -15357.203} C_VEL
LIN {X 0,Y 341.187,Z 423.837,A -85,B 0,C 180,E1 -15358.941,E2 -15358.941} C_VEL
LIN {X 0,Y 340.013,Z 458.246,A -85,B 0,C 180,E1 -15359.703,E2 -15359.703} C_VEL
LIN {X 0,Y 338.961,Z 473.486,A -85,B 0,C 180,E1 -15360.265,E2 -15360.265} C_VEL
LIN {X 0,Y 337.636,Z 488.486,A -85,B 0,C 180,E1 -15361.075,E2 -15361.075} C_VEL
LIN {X 0,Y 336.16,Z 500.879,A -85,B 0,C 180,E1 -15361.939,E2 -15361.939} C_VEL
LIN {X 0,Y 334.183,Z 514.433,A -85,B 0,C 180,E1 -15363.117,E2 -15363.117} C_VEL
LIN {X 0,Y 331.903,Z 528.181,A -85,B 0,C 180,E1 -15364.608,E2 -15364.608} C_VEL
LIN {X 0,Y 329.727,Z 539.519,A -85,B 0,C 180,E1 -15366.11,E2 -15366.11} C_VEL
LIN {X 0,Y 327.541,Z 550.952,A -85,B 0,C 180,E1 -15367.944,E2 -15367.944} C_VEL
LIN {X 0,Y 325.492,Z 560.573,A -85,B 0,C 180,E1 -15369.789,E2 -15369.789} C_VEL
LIN {X 0,Y 323.463,Z 569.997,A -85,B 0,C 180,E1 -15371.963,E2 -15371.963} C_VEL
LIN {X 0,Y 321.784,Z 577.757,A -85,B 0,C 180,E1 -15374.129,E2 -15374.129} C_VEL
LIN {X 0,Y 320.762,Z 583.479,A -85,B 0,C 180,E1 -15376.053,E2 -15376.053} C_VEL
LIN {X 0,Y 319.509,Z 589.631,A -85,B 0,C 180,E1 -15378.581,E2 -15378.581} C_VEL
LIN {X 0,Y 318.709,Z 594.374,A -85,B 0,C 180,E1 -15381.12,E2 -15381.12} C_VEL
LIN {X 0,Y 318.251,Z 597.844,A -85,B 0,C 180,E1 -15383.66,E2 -15383.66} C_VEL
LIN {X 0,Y 317.991,Z 600.137,A -85,B 0,C 180,E1 -15386.198,E2 -15386.198} C_VEL
LIN {X 0,Y 317.852,Z 601.308,A -85,B 0,C 180,E1 -15388.732,E2 -15388.732} C_VEL
LIN {X 0,Y 317.852,Z 601.322,A -85,B 0,C 180,E1 -15391.266,E2 -15391.266} C_VEL
LIN {X 0,Y 317.99,Z 600.209,A -85,B 0,C 180,E1 -15393.801,E2 -15393.801} C_VEL
LIN {X 0,Y 318.286,Z 597.826,A -85,B 0,C 180,E1 -15396.467,E2 -15396.467} C_VEL
LIN {X 0,Y 318.701,Z 594.553,A -85,B 0,C 180,E1 -15398.879,E2 -15398.879} C_VEL
LIN {X 0,Y 319.477,Z 589.868,A -85,B 0,C 180,E1 -15401.419,E2 -15401.419} C_VEL
LIN {X 0,Y 320.7,Z 583.789,A -85,B 0,C 180,E1 -15403.949,E2 -15403.949} C_VEL
LIN {X 0,Y 322.166,Z 576.136,A -85,B 0,C 180,E1 -15406.474,E2 -15406.474} C_VEL
LIN {X 0,Y 323.96,Z 567.964,A -85,B 0,C 180,E1 -15408.662,E2 -15408.662} C_VEL
LIN {X 0,Y 326.046,Z 558.116,A -85,B 0,C 180,E1 -15410.833,E2 -15410.833} C_VEL
LIN {X 0,Y 328.353,Z 546.982,A -85,B 0,C 180,E1 -15412.849,E2 -15412.849} C_VEL
LIN {X 0,Y 330.623,Z 534.873,A -85,B 0,C 180,E1 -15414.655,E2 -15414.655} C_VEL
LIN {X 0,Y 332.936,Z 522.603,A -85,B 0,C 180,E1 -15416.145,E2 -15416.145} C_VEL
LIN {X 0,Y 335.052,Z 509.187,A -85,B 0,C 180,E1 -15417.481,E2 -15417.481} C_VEL
LIN {X 0,Y 336.853,Z 495.278,A -85,B 0,C 180,E1 -15418.591,E2 -15418.591} C_VEL
LIN {X 0,Y 338.491,Z 479.728,A -85,B 0,C 180,E1 -15419.54,E2 -15419.54} C_VEL
LIN {X 0,Y 339.701,Z 464.645,A -85,B 0,C 180,E1 -15420.198,E2 -15420.198} C_VEL
LIN {X 0,Y 340.472,Z 449.045,A -85,B 0,C 180,E1 -15420.636,E2 -15420.636} C_VEL
LIN {X 0,Y 341.033,Z 430.3,A -85,B 0,C 180,E1 -15421.031,E2 -15421.031} C_VEL
LIN {X 0,Y 340.668,Z 424.497,A -85,B 0,C 180,E1 -15421.209,E2 -15421.209} C_VEL
LIN {X 0,Y 336.497,Z 405.836,A -85,B 0,C 180,E1 -15422.105,E2 -15422.105} C_VEL
LIN {X 0,Y 336.103,Z 400.035,A -85,B 0,C 180,E1 -15422.292,E2 -15422.292} C_VEL
LIN {X 0,Y 337.998,Z 342.98,A -85,B 0,C 180,E1 -15423.504,E2 -15423.504} C_VEL
LIN {X 0,Y 329.965,Z 325.552,A -85,B 0,C 180,E1 -15424.894,E2 -15424.894} C_VEL
LIN {X 0,Y 321.821,Z 310.061,A -85,B 0,C 180,E1 -15426.341,E2 -15426.341} C_VEL
LIN {X 0,Y 314.485,Z 298.294,A -85,B 0,C 180,E1 -15427.673,E2 -15427.673} C_VEL
LIN {X 0,Y 312.858,Z 295.7,A -85,B 0,C 180,E1 -15427.98,E2 -15427.98} C_VEL
LIN {X 0,Y 312.489,Z 294.187,A -85,B 0,C 180,E1 -15428.116,E2 -15428.116} C_VEL
LIN {X 0,Y 312.462,Z 294.175,A -85,B 0,C 180,E1 -15432.436,E2 -15432.436} C_VEL
LIN {X 0,Y 312.454,Z 294.186,A -85,B 0,C 180,E1 -15436.035,E2 -15436.035} C_VEL
LIN {X 0,Y 312.452,Z 294.187,A -85,B 0,C 180,E1 -15439.885,E2 -15439.885} C_VEL
LIN {X 0,Y 312.531,Z 294.149,A -85,B 0,C 180,E1 -15444.051,E2 -15444.051} C_VEL
LIN {X 0,Y 312.497,Z 294.183,A -85,B 0,C 180,E1 -15447.333,E2 -15447.333} C_VEL
LIN {X 0,Y 312.481,Z 294.184,A -85,B 0,C 180,E1 -15451.299,E2 -15451.299} C_VEL
LIN {X 0,Y 312.518,Z 294.183,A -85,B 0,C 180,E1 -15454.705,E2 -15454.705} C_VEL
LIN {X 0,Y 312.536,Z 294.173,A -85,B 0,C 180,E1 -15457.525,E2 -15457.525} C_VEL
LIN {X 0,Y 312.542,Z 294.167,A -85,B 0,C 180,E1 -15461.65,E2 -15461.65} C_VEL
LIN {X 0,Y 312.649,Z 294.154,A -85,B 0,C 180,E1 -15465.684,E2 -15465.684} C_VEL
LIN {X 0,Y 312.683,Z 294.157,A -85,B 0,C 180,E1 -15469.641,E2 -15469.641} C_VEL
LIN {X 0,Y 312.793,Z 294.141,A -85,B 0,C 180,E1 -15472.252,E2 -15472.252} C_VEL
LIN {X 0,Y 312.69,Z 294.152,A -85,B 0,C 180,E1 -15474.842,E2 -15474.842} C_VEL
LIN {X 0,Y 312.92,Z 294.127,A -85,B 0,C 180,E1 -15477.425,E2 -15477.425} C_VEL
LIN {X 0,Y 312.979,Z 294.11,A -85,B 0,C 180,E1 -15481.287,E2 -15481.287} C_VEL
LIN {X 0,Y 312.84,Z 294.131,A -85,B 0,C 180,E1 -15486.449,E2 -15486.449} C_VEL
LIN {X 0,Y 312.749,Z 294.15,A -85,B 0,C 180,E1 -15489.05,E2 -15489.05} C_VEL
LIN {X 0,Y 312.633,Z 294.167,A -85,B 0,C 180,E1 -15492.991,E2 -15492.991} C_VEL
LIN {X 0,Y 312.637,Z 294.157,A -85,B 0,C 180,E1 -15495.65,E2 -15495.65} C_VEL
LIN {X 0,Y 312.628,Z 294.161,A -85,B 0,C 180,E1 -15499.236,E2 -15499.236} C_VEL
LIN {X 0,Y 312.541,Z 294.174,A -85,B 0,C 180,E1 -15502.788,E2 -15502.788} C_VEL
LIN {X 0,Y 312.529,Z 294.148,A -85,B 0,C 180,E1 -15505.909,E2 -15505.909} C_VEL
LIN {X 0,Y 312.498,Z 294.179,A -85,B 0,C 180,E1 -15509.655,E2 -15509.655} C_VEL
LIN {X 0,Y 312.518,Z 294.171,A -85,B 0,C 180,E1 -15513.689,E2 -15513.689} C_VEL
LIN {X 0,Y 312.518,Z 294.16,A -85,B 0,C 180,E1 -15517.386,E2 -15517.386} C_VEL
LIN {X 0,Y 312.488,Z 294.183,A -85,B 0,C 180,E1 -15520.709,E2 -15520.709} C_VEL
LIN {X 0,Y 312.449,Z 294.19,A -85,B 0,C 180,E1 -15524.21,E2 -15524.21} C_VEL
LIN {X 0,Y 312.513,Z 294.296,A -85,B 0,C 180,E1 -15527.377,E2 -15527.377} C_VEL
LIN {X 0,Y 316.153,Z 306.301,A -85,B 0,C 180,E1 -15531.081,E2 -15531.081} C_VEL
LIN {X 0,Y 317.694,Z 311.853,A -85,B 0,C 180,E1 -15532.663,E2 -15532.663} C_VEL
LIN {X 0,Y 326.367,Z 329.192,A -85,B 0,C 180,E1 -15534.266,E2 -15534.266} C_VEL
LIN {X 0,Y 333.987,Z 346.14,A -85,B 0,C 180,E1 -15535.625,E2 -15535.625} C_VEL
LIN {X 0,Y 337.271,Z 365.821,A -85,B 0,C 180,E1 -15536.495,E2 -15536.495} C_VEL
LIN {X 0,Y 334.268,Z 458.473,A -85,B 0,C 180,E1 -15538.467,E2 -15538.467} C_VEL
LIN {X 0,Y 333.328,Z 480.997,A -85,B 0,C 180,E1 -15538.987,E2 -15538.987} C_VEL
LIN {X 0,Y 332.103,Z 496.416,A -85,B 0,C 180,E1 -15539.565,E2 -15539.565} C_VEL
LIN {X 0,Y 330.353,Z 511.318,A -85,B 0,C 180,E1 -15540.356,E2 -15540.356} C_VEL
LIN {X 0,Y 328.326,Z 525.77,A -85,B 0,C 180,E1 -15541.385,E2 -15541.385} C_VEL
LIN {X 0,Y 326.181,Z 538.958,A -85,B 0,C 180,E1 -15542.578,E2 -15542.578} C_VEL
LIN {X 0,Y 323.644,Z 552.407,A -85,B 0,C 180,E1 -15544.087,E2 -15544.087} C_VEL
LIN {X 0,Y 321.16,Z 564.663,A -85,B 0,C 180,E1 -15545.776,E2 -15545.776} C_VEL
LIN {X 0,Y 318.781,Z 576.031,A -85,B 0,C 180,E1 -15547.683,E2 -15547.683} C_VEL
LIN {X 0,Y 316.873,Z 585.3,A -85,B 0,C 180,E1 -15549.555,E2 -15549.555} C_VEL
LIN {X 0,Y 314.917,Z 594.589,A -85,B 0,C 180,E1 -15551.794,E2 -15551.794} C_VEL
LIN {X 0,Y 313.135,Z 603.34,A -85,B 0,C 180,E1 -15554.376,E2 -15554.376} C_VEL
LIN {X 0,Y 311.975,Z 610.375,A -85,B 0,C 180,E1 -15556.982,E2 -15556.982} C_VEL
LIN {X 0,Y 311.18,Z 615.912,A -85,B 0,C 180,E1 -15559.591,E2 -15559.591} C_VEL
LIN {X 0,Y 310.806,Z 620.107,A -85,B 0,C 180,E1 -15562.203,E2 -15562.203} C_VEL
LIN {X 0,Y 310.687,Z 623.052,A -85,B 0,C 180,E1 -15564.809,E2 -15564.809} C_VEL
LIN {X 0,Y 310.698,Z 624.809,A -85,B 0,C 180,E1 -15567.408,E2 -15567.408} C_VEL
LIN {X 0,Y 310.758,Z 625.412,A -85,B 0,C 180,E1 -15570.001,E2 -15570.001} C_VEL
LIN {X 0,Y 310.698,Z 624.8,A -85,B 0,C 180,E1 -15572.594,E2 -15572.594} C_VEL
LIN {X 0,Y 310.687,Z 623.03,A -85,B 0,C 180,E1 -15575.192,E2 -15575.192} C_VEL
LIN {X 0,Y 310.804,Z 620.077,A -85,B 0,C 180,E1 -15577.798,E2 -15577.798} C_VEL
LIN {X 0,Y 311.17,Z 615.878,A -85,B 0,C 180,E1 -15580.41,E2 -15580.41} C_VEL
LIN {X 0,Y 311.976,Z 610.326,A -85,B 0,C 180,E1 -15583.02,E2 -15583.02} C_VEL
LIN {X 0,Y 313.136,Z 603.27,A -85,B 0,C 180,E1 -15585.625,E2 -15585.625} C_VEL
LIN {X 0,Y 314.878,Z 594.505,A -85,B 0,C 180,E1 -15588.209,E2 -15588.209} C_VEL
LIN {X 0,Y 316.561,Z 586.656,A -85,B 0,C 180,E1 -15590.129,E2 -15590.129} C_VEL
LIN {X 0,Y 318.835,Z 575.754,A -85,B 0,C 180,E1 -15592.349,E2 -15592.349} C_VEL
LIN {X 0,Y 321.156,Z 564.537,A -85,B 0,C 180,E1 -15594.225,E2 -15594.225} C_VEL
LIN {X 0,Y 323.646,Z 552.257,A -85,B 0,C 180,E1 -15595.914,E2 -15595.914} C_VEL
LIN {X 0,Y 326.187,Z 538.761,A -85,B 0,C 180,E1 -15597.423,E2 -15597.423} C_VEL
LIN {X 0,Y 328.483,Z 524.589,A -85,B 0,C 180,E1 -15598.693,E2 -15598.693} C_VEL
LIN {X 0,Y 330.448,Z 509.873,A -85,B 0,C 180,E1 -15599.724,E2 -15599.724} C_VEL
LIN {X 0,Y 332.255,Z 494.448,A -85,B 0,C 180,E1 -15600.509,E2 -15600.509} C_VEL
LIN {X 0,Y 333.403,Z 479.195,A -85,B 0,C 180,E1 -15601.051,E2 -15601.051} C_VEL
LIN {X 0,Y 336.424,Z 391.302,A -85,B 0,C 180,E1 -15602.94,E2 -15602.94} C_VEL
LIN {X 0,Y 337.216,Z 365.928,A -85,B 0,C 180,E1 -15603.484,E2 -15603.484} C_VEL
LIN {X 0,Y 333.729,Z 345.473,A -85,B 0,C 180,E1 -15604.396,E2 -15604.396} C_VEL
LIN {X 0,Y 324.966,Z 326.337,A -85,B 0,C 180,E1 -15605.957,E2 -15605.957} C_VEL
LIN {X 0,Y 318.913,Z 314.397,A -85,B 0,C 180,E1 -15607.07,E2 -15607.07} C_VEL
LIN {X 0,Y 317.563,Z 311.546,A -85,B 0,C 180,E1 -15607.37,E2 -15607.37} C_VEL
LIN {X 0,Y 314.491,Z 300.767,A -85,B 0,C 180,E1 -15610.553,E2 -15610.553} C_VEL
LIN {X 0,Y 312.49,Z 294.186,A -85,B 0,C 180,E1 -15612.651,E2 -15612.651} C_VEL
LIN {X 0,Y 312.461,Z 294.174,A -85,B 0,C 180,E1 -15616.036,E2 -15616.036} C_VEL
LIN {X 0,Y 312.507,Z 294.179,A -85,B 0,C 180,E1 -15619.875,E2 -15619.875} C_VEL
LIN {X 0,Y 312.538,Z 294.175,A -85,B 0,C 180,E1 -15624.051,E2 -15624.051} C_VEL
LIN {X 0,Y 312.505,Z 294.174,A -85,B 0,C 180,E1 -15627.334,E2 -15627.334} C_VEL
LIN {X 0,Y 312.511,Z 294.175,A -85,B 0,C 180,E1 -15631.292,E2 -15631.292} C_VEL
LIN {X 0,Y 312.552,Z 294.173,A -85,B 0,C 180,E1 -15634.708,E2 -15634.708} C_VEL
LIN {X 0,Y 312.568,Z 294.165,A -85,B 0,C 180,E1 -15637.528,E2 -15637.528} C_VEL
LIN {X 0,Y 312.643,Z 294.159,A -85,B 0,C 180,E1 -15641.657,E2 -15641.657} C_VEL
LIN {X 0,Y 312.699,Z 294.153,A -85,B 0,C 180,E1 -15645.687,E2 -15645.687} C_VEL
LIN {X 0,Y 312.69,Z 294.153,A -85,B 0,C 180,E1 -15649.642,E2 -15649.642} C_VEL
LIN {X 0,Y 312.801,Z 294.138,A -85,B 0,C 180,E1 -15652.253,E2 -15652.253} C_VEL
LIN {X 0,Y 312.693,Z 294.159,A -85,B 0,C 180,E1 -15654.842,E2 -15654.842} C_VEL
LIN {X 0,Y 312.983,Z 294.122,A -85,B 0,C 180,E1 -15658.713,E2 -15658.713} C_VEL
LIN {X 0,Y 312.914,Z 294.128,A -85,B 0,C 180,E1 -15662.575,E2 -15662.575} C_VEL
LIN {X 0,Y 312.843,Z 294.133,A -85,B 0,C 180,E1 -15666.449,E2 -15666.449} C_VEL
LIN {X 0,Y 312.755,Z 294.151,A -85,B 0,C 180,E1 -15669.05,E2 -15669.05} C_VEL
LIN {X 0,Y 312.629,Z 294.167,A -85,B 0,C 180,E1 -15672.991,E2 -15672.991} C_VEL
LIN {X 0,Y 312.572,Z 294.169,A -85,B 0,C 180,E1 -15675.653,E2 -15675.653} C_VEL
LIN {X 0,Y 312.532,Z 294.175,A -85,B 0,C 180,E1 -15679.713,E2 -15679.713} C_VEL
LIN {X 0,Y 312.521,Z 294.173,A -85,B 0,C 180,E1 -15682.776,E2 -15682.776} C_VEL
LIN {X 0,Y 312.485,Z 294.167,A -85,B 0,C 180,E1 -15686.732,E2 -15686.732} C_VEL
LIN {X 0,Y 312.471,Z 294.171,A -85,B 0,C 180,E1 -15689.658,E2 -15689.658} C_VEL
LIN {X 0,Y 312.523,Z 294.178,A -85,B 0,C 180,E1 -15693.688,E2 -15693.688} C_VEL
LIN {X 0,Y 312.513,Z 294.183,A -85,B 0,C 180,E1 -15697.387,E2 -15697.387} C_VEL
LIN {X 0,Y 312.437,Z 294.189,A -85,B 0,C 180,E1 -15700.718,E2 -15700.718} C_VEL
LIN {X 0,Y 312.437,Z 294.187,A -85,B 0,C 180,E1 -15704.212,E2 -15704.212} C_VEL
LIN {X 0,Y 312.419,Z 294.191,A -85,B 0,C 180,E1 -15707.932,E2 -15707.932} C_VEL
LIN {X 0,Y 312.529,Z 294.369,A -85,B 0,C 180,E1 -15712.06,E2 -15712.06} C_VEL
LIN {X 0,Y 313.497,Z 297.019,A -85,B 0,C 180,E1 -15712.274,E2 -15712.274} C_VEL
LIN {X 0,Y 315.195,Z 299.291,A -85,B 0,C 180,E1 -15712.579,E2 -15712.579} C_VEL
LIN {X 0,Y 323.609,Z 313.233,A -85,B 0,C 180,E1 -15714.099,E2 -15714.099} C_VEL
LIN {X 0,Y 333.2,Z 332.348,A -85,B 0,C 180,E1 -15715.788,E2 -15715.788} C_VEL
LIN {X 0,Y 337.839,Z 342.798,A -85,B 0,C 180,E1 -15716.589,E2 -15716.589} C_VEL
LIN {X 0,Y 335.289,Z 420.495,A -85,B 0,C 180,E1 -15718.242,E2 -15718.242} C_VEL
LIN {X 0,Y 333.976,Z 457.373,A -85,B 0,C 180,E1 -15719.052,E2 -15719.052} C_VEL
LIN {X 0,Y 332.872,Z 473.188,A -85,B 0,C 180,E1 -15719.631,E2 -15719.631} C_VEL
LIN {X 0,Y 331.566,Z 487.593,A -85,B 0,C 180,E1 -15720.404,E2 -15720.404} C_VEL
LIN {X 0,Y 329.911,Z 501.156,A -85,B 0,C 180,E1 -15721.359,E2 -15721.359} C_VEL
LIN {X 0,Y 327.875,Z 514.709,A -85,B 0,C 180,E1 -15722.557,E2 -15722.557} C_VEL
LIN {X 0,Y 325.5,Z 528.456,A -85,B 0,C 180,E1 -15724.072,E2 -15724.072} C_VEL
LIN {X 0,Y 323.216,Z 539.795,A -85,B 0,C 180,E1 -15725.597,E2 -15725.597} C_VEL
LIN {X 0,Y 320.967,Z 551.226,A -85,B 0,C 180,E1 -15727.468,E2 -15727.468} C_VEL
LIN {X 0,Y 318.831,Z 560.846,A -85,B 0,C 180,E1 -15729.347,E2 -15729.347} C_VEL
LIN {X 0,Y 316.695,Z 570.271,A -85,B 0,C 180,E1 -15731.564,E2 -15731.564} C_VEL
LIN {X 0,Y 314.853,Z 578.389,A -85,B 0,C 180,E1 -15733.89,E2 -15733.89} C_VEL
LIN {X 0,Y 313.442,Z 585.42,A -85,B 0,C 180,E1 -15736.382,E2 -15736.382} C_VEL
LIN {X 0,Y 312.287,Z 591.217,A -85,B 0,C 180,E1 -15738.971,E2 -15738.971} C_VEL
LIN {X 0,Y 311.688,Z 594.645,A -85,B 0,C 180,E1 -15740.918,E2 -15740.918} C_VEL
LIN {X 0,Y 311.176,Z 598.201,A -85,B 0,C 180,E1 -15743.594,E2 -15743.594} C_VEL
LIN {X 0,Y 310.925,Z 600.407,A -85,B 0,C 180,E1 -15746.111,E2 -15746.111} C_VEL
LIN {X 0,Y 310.763,Z 601.578,A -85,B 0,C 180,E1 -15748.704,E2 -15748.704} C_VEL
LIN {X 0,Y 310.763,Z 601.592,A -85,B 0,C 180,E1 -15751.295,E2 -15751.295} C_VEL
LIN {X 0,Y 310.924,Z 600.478,A -85,B 0,C 180,E1 -15753.888,E2 -15753.888} C_VEL
LIN {X 0,Y 311.191,Z 598.241,A -85,B 0,C 180,E1 -15756.483,E2 -15756.483} C_VEL
LIN {X 0,Y 311.681,Z 594.823,A -85,B 0,C 180,E1 -15759.081,E2 -15759.081} C_VEL
LIN {X 0,Y 312.504,Z 590.138,A -85,B 0,C 180,E1 -15761.677,E2 -15761.677} C_VEL
LIN {X 0,Y 313.767,Z 584.06,A -85,B 0,C 180,E1 -15764.263,E2 -15764.263} C_VEL
LIN {X 0,Y 315.34,Z 576.406,A -85,B 0,C 180,E1 -15766.841,E2 -15766.841} C_VEL
LIN {X 0,Y 317.206,Z 568.234,A -85,B 0,C 180,E1 -15769.074,E2 -15769.074} C_VEL
LIN {X 0,Y 319.392,Z 558.385,A -85,B 0,C 180,E1 -15771.288,E2 -15771.288} C_VEL
LIN {X 0,Y 321.707,Z 547.735,A -85,B 0,C 180,E1 -15773.259,E2 -15773.259} C_VEL
LIN {X 0,Y 323.962,Z 536.245,A -85,B 0,C 180,E1 -15775.026,E2 -15775.026} C_VEL
LIN {X 0,Y 326.346,Z 524.162,A -85,B 0,C 180,E1 -15776.542,E2 -15776.542} C_VEL
LIN {X 0,Y 328.525,Z 511.031,A -85,B 0,C 180,E1 -15777.902,E2 -15777.902} C_VEL
LIN {X 0,Y 330.263,Z 498.512,A -85,B 0,C 180,E1 -15778.954,E2 -15778.954} C_VEL
LIN {X 0,Y 331.995,Z 483.437,A -85,B 0,C 180,E1 -15779.947,E2 -15779.947} C_VEL
LIN {X 0,Y 333.303,Z 468.591,A -85,B 0,C 180,E1 -15780.664,E2 -15780.664} C_VEL
LIN {X 0,Y 334.205,Z 453.865,A -85,B 0,C 180,E1 -15781.143,E2 -15781.143} C_VEL
LIN {X 0,Y 336.103,Z 400.035,A -85,B 0,C 180,E1 -15782.292,E2 -15782.292} C_VEL
LIN {X 0,Y 335.687,Z 394.235,A -85,B 0,C 180,E1 -15782.481,E2 -15782.481} C_VEL
LIN {X 0,Y 331.466,Z 375.627,A -85,B 0,C 180,E1 -15783.425,E2 -15783.425} C_VEL
LIN {X 0,Y 331.159,Z 369.826,A -85,B 0,C 180,E1 -15783.608,E2 -15783.608} C_VEL
LIN {X 0,Y 332.018,Z 345.033,A -85,B 0,C 180,E1 -15784.143,E2 -15784.143} C_VEL
LIN {X 0,Y 324.777,Z 329.298,A -85,B 0,C 180,E1 -15785.441,E2 -15785.441} C_VEL
LIN {X 0,Y 317.207,Z 314.706,A -85,B 0,C 180,E1 -15786.833,E2 -15786.833} C_VEL
LIN {X 0,Y 309.926,Z 303.058,A -85,B 0,C 180,E1 -15788.194,E2 -15788.194} C_VEL
LIN {X 0,Y 307.479,Z 299.22,A -85,B 0,C 180,E1 -15788.67,E2 -15788.67} C_VEL
LIN {X 0,Y 305.951,Z 296.915,A -85,B 0,C 180,E1 -15788.969,E2 -15788.969} C_VEL
LIN {X 0,Y 305.451,Z 295.065,A -85,B 0,C 180,E1 -15789.129,E2 -15789.129} C_VEL
LIN {X 0,Y 305.432,Z 295.049,A -85,B 0,C 180,E1 -15792.581,E2 -15792.581} C_VEL
LIN {X 0,Y 305.418,Z 295.056,A -85,B 0,C 180,E1 -15796.343,E2 -15796.343} C_VEL
LIN {X 0,Y 305.407,Z 295.065,A -85,B 0,C 180,E1 -15799.884,E2 -15799.884} C_VEL
LIN {X 0,Y 305.459,Z 295.029,A -85,B 0,C 180,E1 -15803.637,E2 -15803.637} C_VEL
LIN {X 0,Y 305.462,Z 295.059,A -85,B 0,C 180,E1 -15806.483,E2 -15806.483} C_VEL
LIN {X 0,Y 305.412,Z 295.063,A -85,B 0,C 180,E1 -15809.585,E2 -15809.585} C_VEL
